Omron CX-Programmer project NewProject (CX-Programmer 9.61)

# PLC NewPLC1: CS1H-H CPU64
I/O table (CPU CS1H-CPU64H, CS1W-SCB21-V1): rack 0 slot 3 CS1W-AD081-V1; rack 0 slot 4 CS1W-CT041; rack 0 slot 5 CS1W-CT041; rack 0 slot 6 CS1W-DRM21-V1; rack 0 slot 8 CS1W-CLK21-V1; rack 0 slot 9 CS1W-ETN21(ETN21Mode); rack 1 slot 2 CS1W-MC221(-V1)

## Global symbols (name address type ; comment)
ALL_OK W303.15 BOOL
0.02 BOOL  ; DATA CLEAR
0.04 BOOL  ; CLEAR OF NG WORKPIECE INSULATION TEST
0.05 BOOL  ; CLEAR OF NG WORKPIECE IMPULSE MEASURE
0.06 BOOL  ; CLEAR OF NG WORKPIECE SWING MEASURE
0.07 BOOL  ; CLEAR OF NG WORKPIECE BEARING INSERT
0.08 BOOL  ; CLEAR OF NG WORKPIECE RESISTANCE MEASURE
0.09 BOOL  ; CLEAR OF NG WORKPIECE LENGTH MEASURE
0.10 BOOL  ; CLEAR OF LANE 1 CONFIRMATION THE OPERATION
0.11 BOOL  ; CLEAR OF LANE 2 CONFIRMATION THE OPERATION
0.12 BOOL  ; CLEAR OF ID INVALIDITY OPERATION
1001.04 BOOL  ; AUTO RUNNING (MACHINE No.1)
1001.05 BOOL  ; FAULT STOP AUX (MACHINE No.1)
1001.06 BOOL  ; FAULT STOP (MACHINE No.1)
1002.06 BOOL  ; AUTO RUNNING (MACHINE No.2)
1002.07 BOOL  ; FAULT STOP AUX (MACHINE No.2)
1002.08 BOOL  ; FAULT STOP (MACHINE No.2)
1005.00 BOOL  ; AUTO RUNNING (MACHINE No.3)
1005.01 BOOL  ; FAULT STOP AUX (MACHINE No.3)
1005.02 BOOL  ; FAULT STOP (MACHINE No.3)
1011.00 BOOL  ; AUTO RUNNING (MACHINE No.4)
1011.01 BOOL  ; FAULT STOP AUX (MACHINE No.4)
1011.02 BOOL  ; FAULT STOP (MACHINE No.4)
1011.03 BOOL  ; AUTO RUNNING (MACHINE No.5)
1011.04 BOOL  ; FAULT STOP AUX (MACHINE No.5)
1011.05 BOOL  ; FAULT STOP (MACHINE No.5)
1011.06 BOOL  ; AUTO RUNNING (MACHINE No.6)
1011.07 BOOL  ; FAULT STOP AUX (MACHINE No.6)
1011.08 BOOL  ; FAULT STOP (MACHINE No.6)
1013.04 BOOL  ; AUTO RUNNING (MACHINE No.7)
1013.05 BOOL  ; FAULT STOP AUX (MACHINE No.7)
1013.06 BOOL  ; FAULT STOP (MACHINE No.7)
1015.06 BOOL  ; AUTO RUNNING (MACHINE No.8)
1015.07 BOOL  ; FAULT STOP AUX (MACHINE No.8)
1015.08 BOOL  ; FAULT STOP (MACHINE No.8)
1016.08 BOOL  ; AUTO RUNNING (MACHINE No.9)
1016.09 BOOL  ; FAULT STOP AUX (MACHINE No.9)
1016.10 BOOL  ; FAULT STOP (MACHINE No.9)
1018.00 BOOL  ; CONVEYOR ROTATE FROM FORMER PROCESS
1019.06 BOOL  ; AUTO RUNNING (MACHINE No.10)
1019.07 BOOL  ; FAULT STOP AUX (MACHINE No.10)
1019.08 BOOL  ; FAULT STOP (MACHINE No.10)
1019.11 BOOL  ; from ball caulking mc  PROCESS, UNLOADING ST WORKPIECE NORMAL-TORQUE
1019.12 BOOL  ; From Ball Caulking, UNLOADING ST WORKPIECE NORMAL-TORQUE
1020.01 BOOL  ; ROTATION REQUEST TO FORMER PROCESS
1020.02 BOOL  ; ALL MACHINES SAVING ENERGY OF FLURESCENT LIGHT
1021.00 BOOL  ; AUTO RUNNING (MACHINE No.11)
1021.01 BOOL  ; FAULT STOP AUX (MACHINE No.11)
1021.02 BOOL  ; FAULT STOP (MACHINE No.11)
1200.00 BOOL  ; OFF IN EMERGENCY STOP
1200.01 BOOL  ; OFF IN AUTO STOP
1200.02 BOOL  ; OFF IN CYCLE STOP
1200.03 BOOL  ; OFF IN FAULT STOP
1200.04 BOOL  ; OFF IN TEMPORARY STOP 1
1200.05 BOOL  ; OFF IN STOP WARNING
1200.06 BOOL  ; OFF IN TEMPORARY STOP 2
1200.07 BOOL  ; OFF IN ONLY ALARM
1200.08 BOOL  ; ALARM CALL
1200.09 BOOL  ; STOP WARNING CALL
1200.10 BOOL  ; FORMER/LATTER PROCESS CONDITION WAITING
1200.11 BOOL  ; ALARM ONLY
1200.12 BOOL  ; BUZZER ON 1
1200.13 BOOL  ; ALARM RESET 1
1200.14 BOOL  ; BUZZER ON 2
1200.15 BOOL  ; ALARM RESET 2
1201.00 BOOL  ; UNUSUAL FAULT WITH LAST SCAN
1201.01 BOOL  ; WITH FAULT
1201.02 BOOL  ; ALL CH ENQUIRY COMPLETION
1201.03 BOOL  ; WITH FAULT IN 150CH
1201.04 BOOL  ; WITH FAULT IN 151CH
1201.05 BOOL  ; WITH FAULT IN 152CH
1201.06 BOOL  ; WITH FAULT IN 153CH
1201.07 BOOL  ; WITH FAULT IN 154CH
1201.08 BOOL  ; WITH FAULT IN 155CH
1201.09 BOOL  ; WITH FAULT IN 156CH
1201.10 BOOL  ; WITH FAULT IN 157CH
1201.11 BOOL  ; WITH FAULT IN 158CH
1201.12 BOOL  ; WITH FAULT IN 159CH
1201.13 BOOL  ; ENQUIRY IN PROGRESS WITH FAULT IN CH
1201.14 BOOL  ; WITH FAULT AUXILIARY
1201.15 BOOL  ; FAULT INDICATION CIRCUIT EFFECTIVE
1202.00 BOOL  ; CH EACH FAULT BIT 1
1202.01 BOOL  ; CH EACH FAULT BIT 2
1202.02 BOOL  ; CH EACH FAULT BIT 4
1202.03 BOOL  ; CH EACH FAULT BIT 8
1203.00 BOOL  ; FAULT ENQUIRY IN PROGRESS BIT 00
1203.01 BOOL  ; FAULT ENQUIRY IN PROGRESS BIT 01
1203.02 BOOL  ; FAULT ENQUIRY IN PROGRESS BIT 02
1203.03 BOOL  ; FAULT ENQUIRY IN PROGRESS BIT 03
1203.04 BOOL  ; FAULT ENQUIRY IN PROGRESS BIT 04
1203.05 BOOL  ; FAULT ENQUIRY IN PROGRESS BIT 05
1203.06 BOOL  ; FAULT ENQUIRY IN PROGRESS BIT 06
1203.07 BOOL  ; FAULT ENQUIRY IN PROGRESS BIT 07
1203.08 BOOL  ; FAULT ENQUIRY IN PROGRESS BIT 08
1203.09 BOOL  ; FAULT ENQUIRY IN PROGRESS BIT 09
1203.10 BOOL  ; FAULT ENQUIRY IN PROGRESS BIT 10
1203.11 BOOL  ; FAULT ENQUIRY IN PROGRESS BIT 11
1203.12 BOOL  ; FAULT ENQUIRY IN PROGRESS BIT 12
1203.13 BOOL  ; FAULT ENQUIRY IN PROGRESS BIT 13
1203.14 BOOL  ; FAULT ENQUIRY IN PROGRESS BIT 14
1203.15 BOOL  ; FAULT ENQUIRY IN PROGRESS BIT 15
1204.00 BOOL  ; ENQUIRY IN PROGRESS CH CODE 1
1204.01 BOOL  ; ENQUIRY IN PROGRESS CH CODE 2
1204.02 BOOL  ; ENQUIRY IN PROGRESS CH CODE 4
1204.03 BOOL  ; ENQUIRY IN PROGRESS CH CODE 8
1205.00 BOOL  ; SEARCHING IN FIRST HALF 10CH
1205.01 BOOL  ; SEARCHING IN SECOND HALF 10CH
1205.03 BOOL  ; WITH FAULT IN 160CH
1205.04 BOOL  ; WITH FAULT IN 161CH
1205.05 BOOL  ; WITH FAULT IN 162CH
1205.06 BOOL  ; WITH FAULT IN 163CH
1205.07 BOOL  ; WITH FAULT IN 164CH
1205.08 BOOL  ; WITH FAULT IN 165CH
1205.09 BOOL  ; WITH FAULT IN 166CH
1205.10 BOOL  ; WITH FAULT IN 167CH
1205.11 BOOL  ; WITH FAULT IN 168CH
1205.12 BOOL  ; WITH FAULT IN 169CH
1206.00 BOOL  ; ENQUIRY IN PROGRESS CH CODE 1
1206.01 BOOL  ; ENQUIRY IN PROGRESS CH CODE 2
1206.02 BOOL  ; ENQUIRY IN PROGRESS CH CODE 4
1206.03 BOOL  ; ENQUIRY IN PROGRESS CH CODE 8
1207.00 BOOL  ; FAULT RESET AUXILIARY
1207.01 BOOL  ; FAULT RESET START UP
1207.02 BOOL  ; START UP AUXILIARY
1207.03 BOOL  ; FAULT INDICATION REDUCTION
1208.00 BOOL  ; INDIVIDUAL SELECTION MEMORY
1208.01 BOOL  ; INDIVIDUAL SELECTION MEMORY RELEASE
1208.02 BOOL  ; INDIVIDUAL OPERATION EFFECTIVE AUXILIARY
1208.03 BOOL  ; INDIVIDUAL OPERATION CIRCUIT EFFECTIVE
1208.04 BOOL  ; OPERATION MODE CHANGE PULSE
1208.15 BOOL  ; MASTER ON PULSE
1211.00 BOOL  ; 01ST ALRAM SALL ARIA NO FAULT
1211.01 BOOL  ; 02ST ALRAM SALL ARIA NO FAULT
1211.02 BOOL  ; 03ST ALRAM SALL ARIA NO FAULT
1211.03 BOOL  ; 04ST ALRAM SALL ARIA NO FAULT
1211.04 BOOL  ; 05ST ALRAM SALL ARIA NO FAULT
1211.05 BOOL  ; 06ST ALRAM SALL ARIA NO FAULT
1211.06 BOOL  ; 07ST ALRAM SALL ARIA NO FAULT
1211.07 BOOL  ; 08ST ALRAM SALL ARIA NO FAULT
1211.08 BOOL  ; 09ST ALRAM SALL ARIA NO FAULT
1211.09 BOOL  ; 10ST ALRAM SALL ARIA NO FAULT
1211.10 BOOL  ; 11ST ALRAM SALL ARIA NO FAULT
1211.11 BOOL  ; 12ST ALRAM SALL ARIA NO FAULT
1211.12 BOOL  ; 13ST ALRAM SALL ARIA NO FAULT
1211.13 BOOL  ; 14ST ALRAM SALL ARIA NO FAULT
1211.14 BOOL  ; 15ST ALRAM SALL ARIA NO FAULT
1211.15 BOOL  ; 16ST ALRAM SALL ARIA NO FAULT
1212.00 BOOL  ; 01ST WARNING CALL ARIA NO FAULT
1212.01 BOOL  ; 02ST WARNING CALL ARIA NO FAULT
1212.02 BOOL  ; 03ST WARNING CALL ARIA NO FAULT
1212.03 BOOL  ; 04ST WARNING CALL ARIA NO FAULT
1212.04 BOOL  ; 05ST WARNING CALL ARIA NO FAULT
1212.05 BOOL  ; 06ST WARNING CALL ARIA NO FAULT
1212.06 BOOL  ; 07ST WARNING CALL ARIA NO FAULT
1212.07 BOOL  ; 08ST WARNING CALL ARIA NO FAULT
1212.08 BOOL  ; 09ST WARNING CALL ARIA NO FAULT
1212.09 BOOL  ; 10ST WARNING CALL ARIA NO FAULT
1212.10 BOOL  ; 11ST WARNING CALL ARIA NO FAULT
1212.11 BOOL  ; 12ST WARNING CALL ARIA NO FAULT
1212.12 BOOL  ; 13ST WARNING CALL ARIA NO FAULT
1212.13 BOOL  ; 14ST WARNING CALL ARIA NO FAULT
1212.14 BOOL  ; 15ST WARNING CALL ARIA NO FAULT
1212.15 BOOL  ; 16ST WARNING CALL ARIA NO FAULT
1213.00 BOOL  ; 17ST ALRAM SALL ARIA NO FAULT
1213.01 BOOL  ; 18ST ALRAM SALL ARIA NO FAULT
1213.02 BOOL  ; 19ST ALRAM SALL ARIA NO FAULT
1213.03 BOOL  ; 20ST ALRAM SALL ARIA NO FAULT
1214.00 BOOL  ; 17ST WARNING CALL ARIA NO FAULT
1214.01 BOOL  ; 18ST WARNING CALL ARIA NO FAULT
1214.02 BOOL  ; 19ST WARNING CALL ARIA NO FAULT
1214.03 BOOL  ; 20ST WARNING CALL ARIA NO FAULT
1222.01 BOOL  ; SEQUENCER NORMAL(CS1)
1230.00 BOOL  ; CONVEYOR ON
1235.00 BOOL  ; BEARING SUPPLY ROBOT MOTION PERMIT
1235.01 BOOL  ; BEARING HANGER UPWARD
1235.02 BOOL  ; BEARING SUPPLY ROBOT PROGRAM START
1235.03 BOOL  ; BEARING SUPPLY ROBOT FIXID POSITION RETURN
1235.05 BOOL  ; BEARING SUPPLY ROBOT FIXID POSITION RETURN
1235.06 BOOL  ; BEARING SUPPLY ROBOT TAKING-OUT POSITION START
1235.07 BOOL  ; BEARING TAKE OUT
1235.08 BOOL  ; BEARING SUPPLY ROBOT TAKING-OUT POSITION
1236 CHANNEL  ; BEARING SUPPLY ROBOT OUTPUT
1236.15 BOOL  ; BEARING SUPPLY ROBOT FIXID POSITION
1311.00 BOOL  ; UNLOADING ROBOT GOOD PRODUCT
1350.03 BOOL  ; MASTER SWITCH ON TRIGGER
1350.04 BOOL  ; MASTER SWITCH OFF TRIGGER
1350.11 BOOL  ; X AXIS SETTING SCREEN
1351.08 BOOL  ; FLASH MEMORY PRESERVATION TIMING
1352.00 BOOL  ; FORWARDING PERMISSION
1352.01 BOOL  ; MEMORY DRIVING END
1400.09 BOOL  ; MEMORY WITH SET VALUE CHANGE
1400.10 BOOL  ; WORKPIECE NUMBER CHANGE CHECK
1400.11 BOOL  ; WORKPIECE NUMBER SET UP PB ON
1400.12 BOOL  ; SETTING WORKPIECE NUMBER CHANGE PULSE
1400.13 BOOL  ; SETTING WORKPIECE NUMBER CHANGE
1400.14 BOOL  ; WORKPIECE NUMBER REGISTRATION SCREEN
1400.15 BOOL  ; WORKPIECE NUMBER REGISTRATION SCREEN PULSE
1401.08 BOOL  ; UNDER WORKPIECE NUMBER 1 DISPLAY
1401.09 BOOL  ; UNDER 1 OR LESS WORKPIECE NUMBER DISPLAY
1401.10 BOOL  ; UNDER WORKPIECE NUMBER 9 DISPLAY
1401.11 BOOL  ; UNDER 9 OR MORE WORKPIECE NUMBER DISPLAY
1402.00 BOOL  ; One set display (thickness of core)
1402.01 BOOL  ; One or less is displayed (thickness of core)
1402.02 BOOL  ; Two set display (thickness of core)
1402.03 BOOL  ; Two or less is displayed (thickness of core)
1402.04 BOOL  ; One set display (coil end)
1402.05 BOOL  ; One or less is displayed (coil end)
1402.06 BOOL  ; Two set display (coil end)
1402.07 BOOL  ; Two or less is displayed (coil end)
1402.08 BOOL  ; One set display (bearing insert)
1402.09 BOOL  ; One or less is displayed (bearing insert)
1402.10 BOOL  ; Two set display (bearing insert)
1402.11 BOOL  ; Two or less is displayed (bearing insert)
1403.03 BOOL  ; WITH SET VALUE CHANGE 1
1403.04 BOOL  ; WITH SET VALUE CHANGE 2
1404.01 BOOL  ; Can one product number flow
1404.02 BOOL  ; Can two product number flow
1404.03 BOOL  ; Can three product number flow
1404.04 BOOL  ; Can four product number flow
1404.05 BOOL  ; Can five product number flow
1404.06 BOOL  ; Can six product number flow
1404.07 BOOL  ; Can seven product number flow
1404.08 BOOL  ; Can eight product number flow
1404.09 BOOL  ; Can nine product number flow
1535.00 BOOL  ; The unit is abnormal
1535.06 BOOL  ; Node address repetition
1537.00 BOOL  ; Collation is abnormal
1537.01 BOOL  ; The composition is abnormal
1537.02 BOOL  ; Remote I/O communication abnormality
1537.04 BOOL  ; The scanning list data is illegal
1537.05 BOOL  ; Master function I/O refreshing is abnormal
2000.09 BOOL  ; WITHSTAND VOLTAGE TESTER INTERLOCK
2000.12 BOOL  ; SIGNAL TOWER RED
2000.13 BOOL  ; SIGNAL TOWER YELLOW
2000.14 BOOL  ; SIGNAL TOWER GREEN
2000.15 BOOL  ; ALARM
2001.00 BOOL  ; LOADING CONVEYOR PALLET SHIFT FORWARD
2001.01 BOOL  ; LOADING CONVEYOR PALLET SHIFT BACKWARD
2001.02 BOOL  ; LOADING CONVEYOR PALLET DISCHARGE FORWARD
2001.03 BOOL  ; LOADING CONVEYOR PALLET DISCHARGE BACKWARD
2001.04 BOOL  ; LOADER FORWARD
2001.05 BOOL  ; LOADER BACKWARD
2001.06 BOOL  ; LOADER DOWNWARD
2001.07 BOOL  ; LOADER UPWARD
2001.08 BOOL  ; TURN LOADER CHUCK TURN
2001.09 BOOL  ; TURN LOADER RECHUCK TURN
2001.10 BOOL  ; LOADER CHUCK CLAMP
2001.11 BOOL  ; LOADER CHUCK UNCLAMP
2001.12 BOOL  ; WORKPIECE PUSHER FORWARD
2001.14 BOOL  ; POSITIONING ARROW FORWARD
2002.00 BOOL  ; CONTACT PROBE IN RESISTANCE FORWARD
2002.01 BOOL  ; CONTACT PROBE IN RESISTANCE BACKWARD
2002.02 BOOL  ; CONTACT PROBE IN INPULSE FORWARD
2002.04 BOOL  ; WORKPIECE CLAMP DOWNWARD
2002.05 BOOL  ; WORKPIECE CLAMP UPWARD
2002.06 BOOL  ; TRANSFER CARRIER LIFT UPWARD
2002.07 BOOL  ; TRANSFER CARRIER LIFT DOWNWARD
2002.08 BOOL  ; SUB TRANSFER CARRIER LIFT UPWARD
2002.09 BOOL  ; SUB TRANSFER CARRIER LIFT DOWNWARD
2002.10 BOOL  ; TRANSFER CARRIER FORWARD
2002.11 BOOL  ; TRANSFER CARRIER BACKWARD
2002.12 BOOL  ; LENGTH MEASUREMENT FORWARD
2002.13 BOOL  ; LENGTH MEASUREMENT BACKWARD
2002.14 BOOL  ; Work Clamp DownWard
2002.15 BOOL  ; Work Clamp UpWard
2003.00 BOOL  ; BEARING INSERT (HIGH SPEED) FORWARD
2003.01 BOOL  ; BEARING INSERT (HIGH SPEED) BACKWARD
2003.02 BOOL  ; BEARING INSERT (HIGH PRESSURE) ON
2003.03 BOOL  ; BEARING INSERT (HIGH PRESSURE) OFF
2003.04 BOOL  ; BEARING SHUTTER DOWNWARD
2003.05 BOOL  ; BEARING SHUTTER UPWARD
2003.06 BOOL  ; BEARING GUIDE FORWARD
2003.07 BOOL  ; BEARING GUIDE BACKWARD
2003.08 BOOL  ; BEARING ESCAPE FORWARD
2003.09 BOOL  ; BEARING ESCAPE BACKWARD
2003.10 BOOL  ; BEARING TRANSFER UPWARD
2003.11 BOOL  ; BEARING TRANSFER DOWNWARD
2003.12 BOOL  ; BEARING PUSHER BACKWARD
2003.13 BOOL  ; BEARING PUSHER FORWARD
2003.14 BOOL  ; Work Clamp DownWard
2003.15 BOOL  ; Work Clamp UpWard
2004.00 BOOL  ; BEARING TRANSFER CARRIER FORWARD
2004.01 BOOL  ; BEARING TRANSFER CARRIER BACKWARD
2004.02 BOOL  ; BEARING HANGER FORWARD
2004.03 BOOL  ; BEARING HANGER BACKWARD
2004.04 BOOL  ; BEARING HANGER DOWNWARD
2004.05 BOOL  ; BEARING HANGER UPWARD
2004.06 BOOL  ; UNLOADING ROBOT CHUCK CLAMP
2004.07 BOOL  ; UNLOADING ROBOT CHUCK UNCLAMP
2004.08 BOOL  ; BEARING TRAY ESCAPE FORWARD
2004.09 BOOL  ; BEARING TRAY ESCAPE BACKWARD
2004.10 BOOL  ; BEARING TRAY STOPPER BACKWARD
2004.11 BOOL  ; BEARING TRAY STOPPER FORWARD
2004.12 BOOL  ; BEARING TRAY HOME POSITIONING FORWARD
2004.13 BOOL  ; BEARING TRAY HOME POSITIONING BACKWARD
2004.14 BOOL  ; BEARING TRAY EXCHANGE DOWNWARD
2004.15 BOOL  ; BEARING TRAY EXCHANGE UPWARD
2005.00 BOOL  ; TO RESISTANCE MEASUREMENT_BCD LOWER BYTE OUTPUT
2005.07 BOOL  ; COUNTER
2008.09 BOOL  ; DEFECT DISCHARGING CONVEYOR ON
2008.10 BOOL  ; INVERTER GOOD
2009.00 BOOL  ; LOADING CONVEYOR PALLET SHIFT FORWARD END
2009.01 BOOL  ; LOADING CONVEYOR PALLET SHIFT BACKWARD END
2009.02 BOOL  ; LOADING CONVEYOR PALLET DISCHARGE FORWARD END
2009.03 BOOL  ; LOADING CONVEYOR PALLET DISCHARGE FORWARD END
2009.04 BOOL  ; PALLET ON LOADING CONVEYOR
2009.05 BOOL  ; WORKPIECE ON LOADING CONVEYOR
2010.00 BOOL  ; LOADER FORWARD END
2010.01 BOOL  ; LOADER BACKWARD END
2010.02 BOOL  ; LOADER DOWNWARD END
2010.03 BOOL  ; LOADER UPWARD END
2010.04 BOOL  ; TURN LOADER CHUCK TURN END
2010.05 BOOL  ; TURN LOADER CHUCK RETURN END
2010.07 BOOL  ; LOADER CHUCK UNCLAMP END
2010.08 BOOL  ; PX_ LOADER DOWNWARD END
2010.12 BOOL  ; Contact Probe Lower Resistance Forward
2010.13 BOOL  ; Contact Probe Lower Resistance BackWard
2010.14 BOOL  ; Contact Probe Upper Resistance Forward
2010.15 BOOL  ; Contact Probe Upper Resistance Backward
2011.00 BOOL  ; TRANSFER CARRIER FORWARD END
2011.01 BOOL  ; TRANSFER CARRIER BACKWARD END
2011.02 BOOL  ; TRANSFER CARRIER LIFT UPWARD END
2011.03 BOOL  ; TRANSFER CARRIER LIFT DOWNWARD END
2011.04 BOOL  ; SUB TRANSFER CARRIER LIFT UPWARD END
2011.05 BOOL  ; SUB TRANSFER CARRIER LIFT DOWNWARD END
2011.06 BOOL  ; WORKPIECE PUSHER FORWARD END
2011.07 BOOL  ; WORKPIECE PUSHER BACKWARD END
2011.08 BOOL  ; THICKNESS OF CORE S
2011.09 BOOL  ; THICKNESS OF CORE L
2011.12 BOOL  ; Upper impulse probe forward end
2011.13 BOOL  ; Upper impulse probe receding end
2011.14 BOOL  ; Lower Impulse Probe FWD
2011.15 BOOL  ; Lower impulse probe receding end
2012.00 BOOL  ; POSITIONING ARROW FORWARD END
2012.02 BOOL  ; WORKPIECE CLAMP IN RESISTANCE DOWNWARD END
2012.03 BOOL  ; WORKPIECE CLAMP IN RESISTANCE UPWARD END
2012.04 BOOL  ; WORKPIECE CLAMP IN INPULSE DOWNWARD END
2012.05 BOOL  ; WORKPIECE CLAMP IN INPULSE UPWARD END
2012.06 BOOL  ; CONTACT PROBE IN RESISTANCE FORWARD END
2012.08 BOOL  ; CONTACT PROBE IN INPULSE FORWARD END
2012.10 BOOL  ; CONFIRM POSITIONING
2012.11 BOOL  ; COIL END S
2012.12 BOOL  ; COIL END L
2013.00 BOOL  ; BEARING INSERT (HIGH SPEED) FORWARD END
2013.01 BOOL  ; BEARING INSERT (HIGH SPEED) BACKWARD END
2013.02 BOOL  ; BEARING INSERT (HIGH PRESSURE) ON
2013.04 BOOL  ; BEARING SHUTTER DOWNWARD END
2013.05 BOOL  ; BEARING SHUTTER UPWARD END
2013.06 BOOL  ; BEARING GUIDE FORWARD END
2013.07 BOOL  ; BEARING GUIDE BACKWARD END
2013.08 BOOL  ; BEARING ESCAPE FORWARD END
2013.09 BOOL  ; BEARING ESCAPE BACKWARD END
2013.10 BOOL  ; BEARING TRANSFER UPWARD END
2013.11 BOOL  ; BEARING TRANSFER DOWNWARD END
2013.12 BOOL  ; BEARING PUSHER BACKWARD END
2013.13 BOOL  ; BEARING PUSHER FORWARD END
2013.14 BOOL  ; Bearing press-fit work holding down end
2013.15 BOOL  ; Bearing press-fit work presser rising end
2014.00 BOOL  ; BEARING TRANSFER CARRIER FORWARD END
2014.01 BOOL  ; BEARING TRANSFER CARRIER BACKWARD END
2014.02 BOOL  ; BEARING HANGER FORWARD END
2014.03 BOOL  ; BEARING HANGER BACKWARD END
2014.04 BOOL  ; BEARING HANGER DOWNWARD END
2014.05 BOOL  ; BEARING HANGER UPWARD END
2014.06 BOOL  ; BEARING CHECK (INSIDE AND OUTSIDE)
2014.07 BOOL  ; BEARING CONFIRM
2014.08 BOOL  ; BEARING (BEFOR INSERT)
2014.09 BOOL  ; FULL BEARING
2014.14 BOOL  ; Work Clamp Downword
2014.15 BOOL  ; Work Clamp Upword
2015.00 BOOL  ; LENGTH MEASUREMENT FORWARD END
2015.01 BOOL  ; LENGTH MEASUREMENT BACKWARD END
2015.03 BOOL  ; UNLOADING ROBOT CHUCK UNCLAMP END
2015.04 BOOL  ; WORKPIECE ON DEFECT DISCHARGING CONVEYOR
2015.05 BOOL  ; FULL WORKPIECES ON DEFECT DISCHARGING CONVEYOR
2015.06 BOOL  ; DEFECT DISCHARGING CONVEYOR PAEKING POSITION
2015.07 BOOL  ; CONTAINER
2016.08 BOOL  ; OUT SLAVE 0 FAULT IN COMMUNICATION
2016.09 BOOL  ; OUT SLAVE 1 FAULT IN COMMUNICATION
2016.10 BOOL  ; OUT SLAVE 2 FAULT IN COMMUNICATION
2016.11 BOOL  ; OUT SLAVE 3 FAULT IN COMMUNICATION
2016.12 BOOL  ; OUT SLAVE 4 FAULT IN COMMUNICATION
2016.13 BOOL  ; OUT SLAVE 5 FAULT IN COMMUNICATION
2016.14 BOOL  ; OUT SLAVE 6 FAULT IN COMMUNICATION
2016.15 BOOL  ; OUT SLAVE 7 FAULT IN COMMUNICATION
2017.08 BOOL  ; IN SLAVE 0 FAULT IN COMMUNICATION
2017.09 BOOL  ; IN SLAVE 1 FAULT IN COMMUNICATION
2017.10 BOOL  ; IN SLAVE 2 FAULT IN COMMUNICATION
2017.11 BOOL  ; IN SLAVE 3 FAULT IN COMMUNICATION
2017.12 BOOL  ; IN SLAVE 4 FAULT IN COMMUNICATION
2017.13 BOOL  ; IN SLAVE 5 FAULT IN COMMUNICATION
2017.14 BOOL  ; IN SLAVE 6 FAULT IN COMMUNICATION
2017.15 BOOL  ; IN SLAVE 7 FAULT IN COMMUNICATION
2018.08 BOOL  ; OUT SLAVE 8 FAULT IN COMMUNICATION
2018.09 BOOL  ; OUT SLAVE 9 FAULT IN COMMUNICATION
2018.10 BOOL  ; OUT SLAVE 10 FAULT IN COMMUNICATION
2018.11 BOOL  ; OUT SLAVE 11 FAULT IN COMMUNICATION
2018.12 BOOL  ; OUT SLAVE 12 FAULT IN COMMUNICATION
2018.13 BOOL  ; OUT SLAVE 13 FAULT IN COMMUNICATION
2018.14 BOOL  ; OUT SLAVE 14 FAULT IN COMMUNICATION
2018.15 BOOL  ; OUT SLAVE 15 FAULT IN COMMUNICATION
2019.08 BOOL  ; IN SLAVE 8 FAULT IN COMMUNICATION
2019.09 BOOL  ; IN SLAVE 9 FAULT IN COMMUNICATION
2019.10 BOOL  ; IN SLAVE 10 FAULT IN COMMUNICATION
2019.11 BOOL  ; IN SLAVE 11 FAULT IN COMMUNICATION
2019.12 BOOL  ; IN SLAVE 12 FAULT IN COMMUNICATION
2019.13 BOOL  ; IN SLAVE 13 FAULT IN COMMUNICATION
2019.14 BOOL  ; IN SLAVE 14 FAULT IN COMMUNICATION
2019.15 BOOL  ; IN SLAVE 15 FAULT IN COMMUNICATION
2020.00 BOOL  ; POSITIONING 1 BACKWARD
2020.01 BOOL  ; POSITIONING 1 FORWARD
2020.02 BOOL  ; POSITIONING 2 BACKWARD
2020.03 BOOL  ; POSITIONING 2 FORWARD
2020.04 BOOL  ; ESCAPE BEFOR PALLETIZING UPWARD
2020.05 BOOL  ; ESCAPE BEFOR PALLETIZING DOWNWARD
2020.06 BOOL  ; STOPPER BEFOR PALLETIZING UPWARD
2020.07 BOOL  ; STOPPER BEFOR PALLETIZING DOWNWARD
2020.08 BOOL  ; PALLETIZING STOPPER DOWNWARD
2020.09 BOOL  ; PALLETIZING STOPPER UPWARD
2020.10 BOOL  ; STACKING STOPPER DOWNWARD
2020.11 BOOL  ; STACKING STOPPER UPWARD
2020.12 BOOL  ; UNLOADING ESCAPE UPWARD
2020.13 BOOL  ; UNLOADING ESCAPE DOWNWARD
2020.14 BOOL  ; UNLOADING STOPPER DOWNWARD
2020.15 BOOL  ; UNLOADING STOPPER UPWARD
2021.00 BOOL  ; LIFTER DOWNWARD
2021.01 BOOL  ; LIFTER UPWARD
2021.02 BOOL  ; DROP GUARD BACKWARD
2021.03 BOOL  ; DROP GUARD FORWARD
2021.04 BOOL  ; PALLETIZING LIFTER DOWNWARD
2021.05 BOOL  ; PALLETIZING LIFTER UPWARD
2021.06 BOOL  ; PALLETIZING HOOK BACKWARD
2021.07 BOOL  ; PALLETIZING HOOK FORWARD
2021.08 BOOL  ; STACKING LIFTER DOWNWARD
2021.09 BOOL  ; STACKING LIFTER UPWARD
2021.10 BOOL  ; STACKING HOOK BACKWARD
2021.11 BOOL  ; STACKING HOOK FORWARD
2022.00 BOOL  ; LOADING CONVEYOR
2022.01 BOOL  ; PALLETIZING CONVEYOR
2022.02 BOOL  ; CONVEYOR AFTER PALLETIZING
2022.03 BOOL  ; EXCHANGE CONVEYOR CW
2022.04 BOOL  ; EXCHANGE CONVEYOR CCW
2022.05 BOOL  ; STACKING CONVEYOR
2022.06 BOOL  ; UNLOADING CONVEYOR 1
2022.07 BOOL  ; UNLOADING CONVEYOR 2
2023.00 BOOL  ; POSITIONING 1 BACKWARD
2023.01 BOOL  ; POSITIONING 1 FORWARD
2023.02 BOOL  ; POSITIONING 2 BACKWARD
2023.03 BOOL  ; POSITIONING 2 FORWARD
2023.04 BOOL  ; ESCAPE BEFOR PALLETIZING UPWARD
2023.05 BOOL  ; ESCAPE BEFOR PALLETIZING DOWNWARD
2023.06 BOOL  ; STOPPER BEFOR PALLETIZING UPWARD
2023.07 BOOL  ; STOPPER BEFOR PALLETIZING DOWNWARD
2023.08 BOOL  ; PALLETIZING STOPPER DOWNWARD
2023.09 BOOL  ; PALLETIZING STOPPER UPWARD
2023.10 BOOL  ; STACKING STOPPER DOWNWARD
2023.11 BOOL  ; STACKING STOPPER UPWARD
2023.12 BOOL  ; UNLOADING ESCAPE UPWARD
2023.13 BOOL  ; UNLOADING ESCAPE DOWNWARD
2023.14 BOOL  ; UNLOADING STOPPER DOWNWARD
2023.15 BOOL  ; UNLOADING STOPPER UPWARD
2024.00 BOOL  ; LIFTER DOWNWARD
2024.01 BOOL  ; LIFTER UPWARD
2024.02 BOOL  ; DROP GUARD BACKWARD
2024.03 BOOL  ; DROP GUARD FORWARD
2024.04 BOOL  ; PALLETIZING LIFTER DOWNWARD
2024.05 BOOL  ; PALLETIZING LIFTER UPWARD
2024.06 BOOL  ; PALLETIZING HOOK BACKWARD
2024.07 BOOL  ; PALLETIZING HOOK FORWARD
2024.08 BOOL  ; STACKING LIFTER DOWNWARD
2024.09 BOOL  ; STACKING LIFTER UPWARD
2024.10 BOOL  ; STACKING HOOK BACKWARD
2024.11 BOOL  ; STACKING HOOK FORWARD
2025.00 BOOL  ; LOADING CONVEYOR
2025.01 BOOL  ; PALLETIZING CONVEYOR
2025.02 BOOL  ; CONVEYOR AFTER PALLETIZING
2025.03 BOOL  ; EXCHANGE CONVEYOR CW
2025.04 BOOL  ; EXCHANGE CONVEYOR CCW
2025.05 BOOL  ; STACKING CONVEYOR
2025.06 BOOL  ; UNLOADING CONVEYOR 1
2025.07 BOOL  ; UNLOADING CONVEYOR 2
2028.00 BOOL  ; STOPPER BEFOR PALLETIZING UPWARD END
2028.01 BOOL  ; STOPPER BEFOR PALLETIZING DOWNWARD END
2028.02 BOOL  ; ESCAPE BEFOR PALLETIZING UPWARD END
2028.03 BOOL  ; ESCAPE BEFOR PALLETIZING DOWNWARD END
2028.04 BOOL  ; PALLETIZING STOPPER DOWNWARD END
2028.05 BOOL  ; PALLETIZING STOPPER UPWARD END
2028.06 BOOL  ; PALLETIZING LIFTER 1 DOWNWARD END
2028.07 BOOL  ; PALLETIZING LIFTER 1 INTERMEDIATE POSITION
2028.08 BOOL  ; PALLETIZING LIFTER 1 UPWARD END
2028.09 BOOL  ; PALLETIZING LIFTER 2 DOWNWARD END
2028.10 BOOL  ; PALLETIZING LIFTER 2 INTERMEDIATE POSITION
2028.11 BOOL  ; PALLETIZING LIFTER 2 UPWARD END
2028.12 BOOL  ; PALLETIZING HOOK 1 BACKWARD END
2028.13 BOOL  ; PALLETIZING HOOK 1 FORWARD END
2028.14 BOOL  ; PALLETIZING HOOK 2 BACKWARD END
2028.15 BOOL  ; PALLETIZING HOOK 2 FORWARD END
2029.00 BOOL  ; POSITIONING 2 BACKWARD END
2029.01 BOOL  ; POSITIONING 2 FORWARD END
2029.02 BOOL  ; POSITIONING 1 BACKWARD END
2029.03 BOOL  ; POSITIONING 1 FORWARD END
2029.04 BOOL  ; LOADING CONTAINER
2029.05 BOOL  ; CONTAINER BEFOR PALLETIZING
2029.06 BOOL  ; PALLETIZING CONTAINER
2029.07 BOOL  ; PALLETIZING CONTAINER UPPER SECTION
2029.08 BOOL  ; CONTAINER BEFOR EXCHANGE
2029.09 BOOL  ; EXCHANGE CONTAINER
2030.00 BOOL  ; LIFTER DOWNWARD END
2030.01 BOOL  ; LIFTER UPWARD END
2030.02 BOOL  ; DROP GUARD BACKWARD END
2030.03 BOOL  ; DROP GUARD FORWARD END
2030.04 BOOL  ; STACKING LIFTER 1 DOWNWARD END
2030.05 BOOL  ; STACKING LIFTER 1 INTERMEDIATE POSITION
2030.06 BOOL  ; STACKING LIFTER 1 UPWARD END
2030.07 BOOL  ; STACKING LIFTER 2 DOWNWARD END
2030.08 BOOL  ; STACKING LIFTER 2 INTERMEDIATE POSITION
2030.09 BOOL  ; STACKING LIFTER 2 UPWARD END
2030.10 BOOL  ; STACKING HOOK 1 BACKWARD END
2030.11 BOOL  ; STACKING HOOK 1 FORWARD END
2030.12 BOOL  ; STACKING HOOK 2 BACKWARD END
2030.13 BOOL  ; STACKING HOOK 2 FORWARD END
2030.14 BOOL  ; STACKING STOPPER DOWNWARD END
2030.15 BOOL  ; STACKING STOPPER UPWARD END
2031.00 BOOL  ; UNLOADING ESCAPE UPWARD END
2031.01 BOOL  ; UNLOADING ESCAPE DOWNWARD END
2031.02 BOOL  ; UNLOADING STOPPER DOWNWARD END
2031.03 BOOL  ; UNLOADING STOPPER UPWARD END
2031.04 BOOL  ; PASSING EXCHANGE CONTAINER
2031.05 BOOL  ; STACKING CONTAINER UPPER SECTION
2031.06 BOOL  ; STACKING CONTAINER
2031.07 BOOL  ; FULL CONTAINERS ON UNLOADING CONVEYOR
2031.08 BOOL  ; UNLOADING CONTAINERS
2032.00 BOOL  ; STOPPER BEFOR PALLETIZING UPWARD END
2032.01 BOOL  ; STOPPER BEFOR PALLETIZING DOWNWARD END
2032.02 BOOL  ; ESCAPE BEFOR PALLETIZING UPWARD END
2032.03 BOOL  ; ESCAPE BEFOR PALLETIZING DOWNWARD END
2032.04 BOOL  ; PALLETIZING STOPPER DOWNWARD END
2032.05 BOOL  ; PALLETIZING STOPPER UPWARD END
2032.06 BOOL  ; PALLETIZING LIFTER 1 DOWNWARD END
2032.07 BOOL  ; PALLETIZING LIFTER 1 INTERMEDIATE POSITION
2032.08 BOOL  ; PALLETIZING LIFTER 1 UPWARD END
2032.09 BOOL  ; PALLETIZING LIFTER 2 DOWNWARD END
2032.10 BOOL  ; PALLETIZING LIFTER 2 INTERMEDIATE POSITION
2032.11 BOOL  ; PALLETIZING LIFTER 2 UPWARD END
2032.12 BOOL  ; PALLETIZING HOOK 1 BACKWARD END
2032.13 BOOL  ; PALLETIZING HOOK 1 FORWARD END
2032.14 BOOL  ; PALLETIZING HOOK 2 BACKWARD END
2032.15 BOOL  ; PALLETIZING HOOK 2 FORWARD END
2033.00 BOOL  ; POSITIONING 2 BACKWARD END
2033.01 BOOL  ; POSITIONING 2 FORWARD END
2033.02 BOOL  ; POSITIONING 1 BACKWARD END
2033.03 BOOL  ; POSITIONING 1 FORWARD END
2033.04 BOOL  ; LOADING CONTAINER
2033.05 BOOL  ; CONTAINER BEFOR PALLETIZING
2033.06 BOOL  ; PALLETIZING CONTAINER
2033.07 BOOL  ; PALLETIZING CONTAINER UPPER SECTION
2033.08 BOOL  ; CONTAINER BEFOR EXCHANGE
2033.09 BOOL  ; EXCHANGE CONTAINER
2034.00 BOOL  ; LIFTER DOWNWARD END
2034.01 BOOL  ; LIFTER UPWARD END
2034.02 BOOL  ; DROP GUARD BACKWARD END
2034.03 BOOL  ; DROP GUARD FORWARD END
2034.04 BOOL  ; STACKING LIFTER 1 DOWNWARD END
2034.05 BOOL  ; STACKING LIFTER 1 INTERMEDIATE POSITION
2034.06 BOOL  ; STACKING LIFTER 1 UPWARD END
2034.07 BOOL  ; STACKING LIFTER 2 DOWNWARD END
2034.08 BOOL  ; STACKING LIFTER 2 INTERMEDIATE POSITION
2034.09 BOOL  ; STACKING LIFTER 2 UPWARD END
2034.10 BOOL  ; STACKING HOOK 1 BACKWARD END
2034.11 BOOL  ; STACKING HOOK 1 FORWARD END
2034.12 BOOL  ; STACKING HOOK 2 BACKWARD END
2034.13 BOOL  ; STACKING HOOK 2 FORWARD END
2034.14 BOOL  ; STACKING STOPPER DOWNWARD END
2034.15 BOOL  ; STACKING STOPPER UPWARD END
2035.00 BOOL  ; UNLOADING ESCAPE UPWARD END
2035.01 BOOL  ; UNLOADING ESCAPE DOWNWARD END
2035.02 BOOL  ; UNLOADING STOPPER DOWNWARD END
2035.03 BOOL  ; UNLOADING STOPPER UPWARD END
2035.04 BOOL  ; PASSING EXCHANGE CONTAINER
2035.05 BOOL  ; STACKING CONTAINER UPPER SECTION
2035.06 BOOL  ; STACKING CONTAINER
2035.07 BOOL  ; FULL CONTAINERS ON UNLOADING CONVEYOR
2035.08 BOOL  ; UNLOADING CONTAINERS
2036.08 BOOL  ; OUT SLAVE 0 FAULT IN COMMUNICATION
2036.09 BOOL  ; OUT SLAVE 1 FAULT IN COMMUNICATION
2036.10 BOOL  ; OUT SLAVE 2 FAULT IN COMMUNICATION
2036.11 BOOL  ; OUT SLAVE 3 FAULT IN COMMUNICATION
2036.12 BOOL  ; OUT SLAVE 4 FAULT IN COMMUNICATION
2036.13 BOOL  ; OUT SLAVE 5 FAULT IN COMMUNICATION
2036.14 BOOL  ; OUT SLAVE 6 FAULT IN COMMUNICATION
2036.15 BOOL  ; OUT SLAVE 7 FAULT IN COMMUNICATION
2037.08 BOOL  ; IN SLAVE 0 FAULT IN COMMUNICATION
2037.09 BOOL  ; IN SLAVE 1 FAULT IN COMMUNICATION
2037.10 BOOL  ; IN SLAVE 2 FAULT IN COMMUNICATION
2037.11 BOOL  ; IN SLAVE 3 FAULT IN COMMUNICATION
2037.12 BOOL  ; IN SLAVE 4 FAULT IN COMMUNICATION
2037.13 BOOL  ; IN SLAVE 5 FAULT IN COMMUNICATION
2037.14 BOOL  ; IN SLAVE 6 FAULT IN COMMUNICATION
2037.15 BOOL  ; IN SLAVE 7 FAULT IN COMMUNICATION
2038.08 BOOL  ; OUT SLAVE 8 FAULT IN COMMUNICATION
2038.09 BOOL  ; OUT SLAVE 9 FAULT IN COMMUNICATION
2038.10 BOOL  ; OUT SLAVE 10 FAULT IN COMMUNICATION
2038.11 BOOL  ; OUT SLAVE 11 FAULT IN COMMUNICATION
2038.12 BOOL  ; OUT SLAVE 12 FAULT IN COMMUNICATION
2038.13 BOOL  ; OUT SLAVE 13 FAULT IN COMMUNICATION
2038.14 BOOL  ; OUT SLAVE 14 FAULT IN COMMUNICATION
2038.15 BOOL  ; OUT SLAVE 15 FAULT IN COMMUNICATION
2039.08 BOOL  ; IN SLAVE 8 FAULT IN COMMUNICATION
2039.09 BOOL  ; IN SLAVE 9 FAULT IN COMMUNICATION
2039.10 BOOL  ; IN SLAVE 10 FAULT IN COMMUNICATION
2039.11 BOOL  ; IN SLAVE 11 FAULT IN COMMUNICATION
2039.12 BOOL  ; IN SLAVE 12 FAULT IN COMMUNICATION
2039.13 BOOL  ; IN SLAVE 13 FAULT IN COMMUNICATION
2039.14 BOOL  ; IN SLAVE 14 FAULT IN COMMUNICATION
2039.15 BOOL  ; IN SLAVE 15 FAULT IN COMMUNICATION
2040.00 BOOL  ; DEFECT DISCHARGING CONVEYOR START
2040.01 BOOL  ; DEFECT DISCHARGING CONVEYOR HIGH SPEED
2040.04 BOOL  ; DRIVE WORKPIECE
2040.05 BOOL  ; DRIVE WORKPIECE
2040.09 BOOL  ; FLURESCENT LIGHT OFF
2040.10 BOOL  ; DEFECT DISCHARGING CONVEYOR ON
2040.11 BOOL  ; LANE 1 UNLOADING
2040.12 BOOL  ; LANE 2 UNLOADING
2040.15 BOOL  ; Imagerogar 1
2041 CHANNEL  ; COMMAND POSITION
2041.00 BOOL  ; BEARING SUPPLY ROBOT HOLD
2041.01 BOOL  ; BEARING SUPPLY ROBOT SERVO ON
2041.02 BOOL  ; BEARING SUPPLY ROBOT RESET
2041.03 BOOL  ; BEARING SUPPLY ROBOT START
2042.00 BOOL  ; EXCHANGE CONVEYOR CW ROTATE
2042.01 BOOL  ; EXCHANGE CONVEYOR CCW ROTATE
2042.02 BOOL  ; LOADING CONVEYOR ON
2042.03 BOOL  ; UNLOADING CONVEYOR ON
2042.05 BOOL  ; Resistance Meas. Change Relay 6
2042.06 BOOL  ; Resistance Meas. Change Relay 12
2042.07 BOOL  ; Resistance Meas. Change Relay 13
2042.08 BOOL  ; Resistance Meas. Change Relay 13
2042.09 BOOL  ; Resistance Meas. Change Relay 14
2042.10 BOOL  ; Resistance Meas. Change Relay 15
2042.11 BOOL  ; Resistance Meas. Change Relay 16
2042.12 BOOL  ; Resistance Meas. Change Relay 16
2042.13 BOOL  ; Resistance Meas. Change Relay 17
2042.14 BOOL  ; Resistance Meas. Change Relay 15
2042.15 BOOL  ; Resistance Meas. Change Relay 2
2043.00 BOOL  ; WITH.VOL.MEAS. START
2043.01 BOOL  ; WITH.VOL.MEAS. STOP
2043.02 BOOL  ; RESISTANCE MEAS. TRIG
2043.09 BOOL  ; COUNTER
2043.10 BOOL  ; INPULSE DISPLAY OFF
2043.11 BOOL  ; INPULSE MEAS. START
2043.12 BOOL  ; INPULSE MEAS. RESET
2043.13 BOOL  ; INPULSE TRIG SIGNAL
2044 CHANNEL  ; IMPULSE TESTER
2044.09 BOOL  ; COUNTER
2045 CHANNEL  ; Impulse switching relay
2045.00 BOOL  ; WITHSTAND CIRCUIT CONNECTION
2045.01 BOOL  ; CONDUCTOT CHECK
2046 CHANNEL  ; IMPULSE RELAY
2047 CHANNEL  ; RESISTANCE MEASUREMENT CHANGE RELAY
2047.00 BOOL  ; Resistance Meas. Change Relay 1
2047.01 BOOL  ; Resistance Meas. Change Relay 2
2047.02 BOOL  ; Resistance Meas. Change Relay 3
2047.03 BOOL  ; Resistance Meas. Change Relay 4
2047.04 BOOL  ; Resistance Meas. Change Relay 5
2047.05 BOOL  ; Resistance Meas. Change Relay 6
2047.06 BOOL  ; Resistance Meas. Change Relay 7
2047.07 BOOL  ; Resistance Meas. Change Relay 8
2047.08 BOOL  ; Resistance Meas. Change Relay 9
2047.09 BOOL  ; Resistance Meas. Change Relay 10
2047.10 BOOL  ; Resistance Meas. Change Relay 11
2047.11 BOOL  ; Resistance Meas. Change Relay 12
2047.12 BOOL  ; Resistance Meas. Change Relay 13
2047.13 BOOL  ; Resistance Meas. Change Relay 14
2047.14 BOOL  ; Turn Number Description Switching Relay 1
2047.15 BOOL  ; Turn Number Description Switching Relay 1
2048.00 BOOL  ; INVERTER 2 GOOD
2048.02 BOOL  ; LANE 1 UNLOADING START
2048.03 BOOL  ; ﾚｰﾝ2排出部起動PB
2048.05 BOOL  ; ROBOT CPU GOOD
2048.06 BOOL  ; LANE 1 UNLOADING START
2048.07 BOOL  ; LANE 2 UNLOADING START
2048.08 BOOL  ; DEFECT DISCHARGING CONVEYOR START
2048.09 BOOL  ; ADD SENSOR CHECK BEARING
2049 CHANNEL  ; BEARING SUPPLY ROBOT OUTPUT
2049.00 BOOL  ; BEARING SUPPLY ROBOT MOTION
2049.02 BOOL  ; BEARING SUPPLY ROBOT ALARM
2049.04 BOOL  ; BEARING SUPPLY ROBOT HOMING COMPLETE
2049.05 BOOL  ; BEARING SUPPLY ROBOT POSITIONING COMPLETE
2049.06 BOOL  ; BEARING SUPPLY ROBOT SERVO ON
2051 CHANNEL  ; RESISTANCE MEASUREMENT DATA BCD
2051.00 BOOL  ; RESISTANCE MEASURED VALUE BCD4-0/RNG_OUT0
2051.01 BOOL  ; RESISTANCE MEASURED VALUE BCD4-1 /RNG_OUT1
2051.02 BOOL  ; RESISTANCE MEASURED VALUE BCD4-2 /RNG_OUT2
2051.03 BOOL  ; RESISTANCE MEASURED VALUE BCD4-3 /RNG_OUT3
2051.04 BOOL  ; RESISTANCE MEASURED VALUE BCD5/BCD1-0
2051.05 BOOL  ; RESISTANCE MEASURED VALUE BCD5/BCD1-1
2051.06 BOOL  ; RESISTANCE MEASURED VALUE BCD5/BCD1-2
2051.07 BOOL  ; RESISTANCE MEASURED VALUE BCD5/BCD1-3
2051.08 BOOL  ; RESISTANCE MEASURED VALUE BCD6/BCD2-0
2051.09 BOOL  ; RESISTANCE MEASURED VALUE BCD6/BCD2-1
2051.10 BOOL  ; RESISTANCE MEASURED VALUE BCD6/BCD2-2
2051.11 BOOL  ; RESISTANCE MEASURED VALUE BCD6/BCD2-3
2051.12 BOOL  ; RESISTANCE MEASURED VALUE BCD7/BCD3-0
2051.13 BOOL  ; RESISTANCE MEASURED VALUE BCD7/BCD3-1
2051.14 BOOL  ; RESISTANCE MEASURED VALUE BCD7/BCD3-2
2051.15 BOOL  ; RESISTANCE MEASURED VALUE BCD7/BCD3-3
2052 CHANNEL  ; RESISTANCE MEASUREMENT DATA BCD
2052.05 BOOL  ; RESISTANCE MEAS.1 ERR
2052.06 BOOL  ; RESISTANCE MEAS.1 INDEX
2052.07 BOOL  ; RESISTANCE MEAS.1 EOC
2052.08 BOOL  ; RESISTANCE MEAS.1 BCD 10^4X1
2052.09 BOOL  ; RESISTANCE MEAS.1 BCD 10^4X2
2052.10 BOOL  ; RESISTANCE MEAS.1 BCD 10^4X4
2052.13 BOOL  ; RESISTANCE MEAS.1 BCD 10^5X2
2052.14 BOOL  ; RESISTANCE MEAS.1 BCD 10^5X4
2052.15 BOOL  ; RESISTANCE MEAS.1 BCD 10^5X8
2053.00 BOOL  ; WITH.VOL.TEST
2053.01 BOOL  ; WITH.VOL.OK
2053.02 BOOL  ; WITH.VOL.HIGH-FAULT
2053.03 BOOL  ; WITH.VOL.LOW-FAULT
2053.04 BOOL  ; WITH.VOL.READY
2053.05 BOOL  ; WITH.VOL.PROTECTION
2053.06 BOOL  ; $?St$Bk?_#[5] / NUMBER OF TURNS "HI"$?St$Bk?_#[5]
2053.07 BOOL  ; $?St$Bk?_#[6] / NUMBER OF TURNS "IN"$?St$Bk?_#[6]
2053.08 BOOL  ; $?St$Bk?_#[7] / NUMBER OF TURNS "LO"$?St$Bk?_#[7]
2053.09 BOOL  ; EOM
2053.12 BOOL  ; INPULSE TESTER 1 BUSY
2053.13 BOOL  ; INPULSE TESTER 1 OK
2053.14 BOOL  ; INPULSE TESTER 1 NG
2053.15 BOOL  ; INPULSE TESTER 1 ERROR
2056.08 BOOL  ; OUT SLAVE 0 FAULT IN COMMUNICATION
2056.09 BOOL  ; OUT SLAVE 1 FAULT IN COMMUNICATION
2056.10 BOOL  ; OUT SLAVE 2 FAULT IN COMMUNICATION
2056.11 BOOL  ; OUT SLAVE 3 FAULT IN COMMUNICATION
2056.12 BOOL  ; OUT SLAVE 4 FAULT IN COMMUNICATION
2056.13 BOOL  ; OUT SLAVE 5 FAULT IN COMMUNICATION
2056.14 BOOL  ; OUT SLAVE 6 FAULT IN COMMUNICATION
2056.15 BOOL  ; OUT SLAVE 7 FAULT IN COMMUNICATION
2057.08 BOOL  ; IN SLAVE 0 FAULT IN COMMUNICATION
2057.09 BOOL  ; IN SLAVE 1 FAULT IN COMMUNICATION
2057.10 BOOL  ; IN SLAVE 2 FAULT IN COMMUNICATION
2057.11 BOOL  ; IN SLAVE 3 FAULT IN COMMUNICATION
2057.12 BOOL  ; IN SLAVE 4 FAULT IN COMMUNICATION
2057.13 BOOL  ; IN SLAVE 5 FAULT IN COMMUNICATION
2057.14 BOOL  ; IN SLAVE 6 FAULT IN COMMUNICATION
2057.15 BOOL  ; IN SLAVE 7 FAULT IN COMMUNICATION
2058.08 BOOL  ; OUT SLAVE 8 FAULT IN COMMUNICATION
2058.09 BOOL  ; OUT SLAVE 9 FAULT IN COMMUNICATION
2058.10 BOOL  ; OUT SLAVE 10 FAULT IN COMMUNICATION
2058.11 BOOL  ; OUT SLAVE 11 FAULT IN COMMUNICATION
2058.12 BOOL  ; OUT SLAVE 12 FAULT IN COMMUNICATION
2058.13 BOOL  ; OUT SLAVE 13 FAULT IN COMMUNICATION
2058.14 BOOL  ; OUT SLAVE 14 FAULT IN COMMUNICATION
2058.15 BOOL  ; OUT SLAVE 15 FAULT IN COMMUNICATION
2059.08 BOOL  ; IN SLAVE 8 FAULT IN COMMUNICATION
2059.09 BOOL  ; IN SLAVE 9 FAULT IN COMMUNICATION
2059.10 BOOL  ; IN SLAVE 10 FAULT IN COMMUNICATION
2059.11 BOOL  ; IN SLAVE 11 FAULT IN COMMUNICATION
2059.12 BOOL  ; IN SLAVE 12 FAULT IN COMMUNICATION
2059.13 BOOL  ; IN SLAVE 13 FAULT IN COMMUNICATION
2059.14 BOOL  ; IN SLAVE 14 FAULT IN COMMUNICATION
2059.15 BOOL  ; IN SLAVE 15 FAULT IN COMMUNICATION
2061 CHANNEL  ; INPUT 1 CONVERSION VALUE
2069.00 BOOL  ; INPUT 1 DISCONNECTION DETECTION
2080.00 BOOL  ; MASTER ON PERMISSION
2080.01 BOOL  ; SAFETY DOOR OPEN OK(FROM PLC)
2080.02 BOOL  ; CONVEYOR ON PERMISSION
2080.03 BOOL  ; CONVEYOR ECO RUNNING 1
2080.04 BOOL  ; MASTER SWITCH ON
2080.05 BOOL  ; CONVEYOR SWITCH ON
2080.06 BOOL  ; CONVEYOR ECO RUNNING 2
2080.07 BOOL  ; ROBOT STOP FROM PLC(AT OFF)
2088.00 BOOL  ; BEARING TRAY EXCHANGE DOWNWARD END
2088.01 BOOL  ; BEARING TRAY EXCHANGE UPWARD END
2088.02 BOOL  ; BEARING TRAY HOME POSITIONING BACKWARD END
2088.03 BOOL  ; BEARING TRAY HOME POSITIONING FORWARD END
2088.04 BOOL  ; BEARING TRAY STOPPER BACKWARD END
2088.05 BOOL  ; BEARING TRAY STOPPER FORWARD END
2088.06 BOOL  ; BEARING TRAY ESCAPE FORWARD END
2088.07 BOOL  ; BEARING TRAY ESCAPE BACKWARD END
2088.08 BOOL  ; LOADING BEARING TRAY
2088.09 BOOL  ; BEARING TRAY BEFOR EXCHANGE
2088.10 BOOL  ; EXCHANGE BEARING TRAY
2088.11 BOOL  ; PASSING BEARING TRAY
2088.12 BOOL  ; PASSING UNLOADING BEARING TRAY
2090.00 BOOL  ; FUSE GOOD
2090.01 BOOL  ; THERMAL RELAY GOOD
2090.02 BOOL  ; SAFETY CONFIRM 1-1(SAFETY DOOR SWITCH 1 CLOSE WHEN TEACHING ROBOT)
2090.03 BOOL  ; EX. HANDLE CONFIRMATION
2090.04 BOOL  ; SAFETY CONFIRM 2-1(SAFETY DOOR SWITCH 1 OPEN WHEN TEACHING ROBOT)
2090.05 BOOL  ; AIR CONFIRMATION
2090.06 BOOL  ; CONVEYOR THERMAL RELAY GOOD
2090.07 BOOL  ; MASTER ON CONFIRM
2090.08 BOOL  ; CONVEYOR ON CONFIRM
2090.09 BOOL  ; SAFETY CONFIRM 1-2(SAFETY DOOR SWITCH 2 CLOSE WHEN TEACHING ROBOT)
2090.10 BOOL  ; SAFETY CONFIRM 2-2(SAFETY DOOR SWITCH 2 OPEN WHEN TEACHING ROBOT)
2090.11 BOOL  ; SAFTY CONFIRM INVALID(KEY SWITCH TEACH ON)
2090.12 BOOL  ; EMERGENCY STOP PUSH BUTTON SWITCH OFF
2090.13 BOOL  ; SAFTY CONFIRM INVALID PL
2090.14 BOOL  ; MASTER ON COND.(EXT. A SAFEGUARD)
2090.15 BOOL  ; OPERATION PANEL SURE PUSH BUTTON SWITCH
2091.07 BOOL  ; MASTER ON CONFIRM MC-A
2091.15 BOOL  ; OPERATION PANEL SURE PUSH BUTTON SWITCH CR-A
2096.08 BOOL  ; OUT SLAVE 0 FAULT IN COMMUNICATION
2096.09 BOOL  ; OUT SLAVE 1 FAULT IN COMMUNICATION
2096.10 BOOL  ; OUT SLAVE 2 FAULT IN COMMUNICATION
2096.11 BOOL  ; OUT SLAVE 3 FAULT IN COMMUNICATION
2096.12 BOOL  ; OUT SLAVE 4 FAULT IN COMMUNICATION
2096.13 BOOL  ; OUT SLAVE 5 FAULT IN COMMUNICATION
2096.14 BOOL  ; OUT SLAVE 6 FAULT IN COMMUNICATION
2096.15 BOOL  ; OUT SLAVE 7 FAULT IN COMMUNICATION
2097.08 BOOL  ; IN SLAVE 0 FAULT IN COMMUNICATION
2097.09 BOOL  ; IN SLAVE 1 FAULT IN COMMUNICATION
2097.10 BOOL  ; IN SLAVE 2 FAULT IN COMMUNICATION
2097.11 BOOL  ; IN SLAVE 3 FAULT IN COMMUNICATION
2097.12 BOOL  ; IN SLAVE 4 FAULT IN COMMUNICATION
2097.13 BOOL  ; IN SLAVE 5 FAULT IN COMMUNICATION
2097.14 BOOL  ; IN SLAVE 6 FAULT IN COMMUNICATION
2097.15 BOOL  ; IN SLAVE 7 FAULT IN COMMUNICATION
2098.08 BOOL  ; OUT SLAVE 8 FAULT IN COMMUNICATION
2098.09 BOOL  ; OUT SLAVE 9 FAULT IN COMMUNICATION
2098.10 BOOL  ; OUT SLAVE 10 FAULT IN COMMUNICATION
2098.11 BOOL  ; OUT SLAVE 11 FAULT IN COMMUNICATION
2098.12 BOOL  ; OUT SLAVE 12 FAULT IN COMMUNICATION
2098.13 BOOL  ; OUT SLAVE 13 FAULT IN COMMUNICATION
2098.14 BOOL  ; OUT SLAVE 14 FAULT IN COMMUNICATION
2098.15 BOOL  ; OUT SLAVE 15 FAULT IN COMMUNICATION
2099.08 BOOL  ; IN SLAVE 8 FAULT IN COMMUNICATION
2099.09 BOOL  ; IN SLAVE 9 FAULT IN COMMUNICATION
2099.10 BOOL  ; IN SLAVE 10 FAULT IN COMMUNICATION
2099.11 BOOL  ; IN SLAVE 11 FAULT IN COMMUNICATION
2099.12 BOOL  ; IN SLAVE 12 FAULT IN COMMUNICATION
2099.13 BOOL  ; IN SLAVE 13 FAULT IN COMMUNICATION
2099.14 BOOL  ; IN SLAVE 14 FAULT IN COMMUNICATION
2099.15 BOOL  ; IN SLAVE 15 FAULT IN COMMUNICATION
2100.00 BOOL  ; $?St$Bk?_#[8] / Brake / Output $?St$Bk?_#[8]
2100.14 BOOL  ; Error Reset Bit
2101.01 BOOL  ; OPTIONAL INPUT # 1
2101.02 BOOL  ; OPTIONAL INPUT # 2
2102 CHANNEL  ; Task 1 program number
2103.01 BOOL  ; Automatic/Manual Mode ↑
2103.02 BOOL  ; Cycle Start Bit
2103.03 BOOL  ; Single Block
2103.04 BOOL  ; Forced Block End
2103.05 BOOL  ; Pause
2103.06 BOOL  ; M Code Reset Bit
2103.07 BOOL  ; $?St$Bk?_#[9] / Program Number Read / Bit$?St$Bk?_#[9]
2103.09 BOOL  ; Teaching Bit
2103.10 BOOL  ; Teaching Type Bit
2106 CHANNEL  ; X AXIS OVERRIDE
2107.00 BOOL  ; Deceleration Stop
2107.01 BOOL  ; Origin Search
2107.02 BOOL  ; Reference Origin Return
2107.03 BOOL  ; Jogging
2107.04 BOOL  ; Error Counter Reset
2107.05 BOOL  ; Forced Origin
2107.06 BOOL  ; Absolute Origin Set
2107.08 BOOL  ; $?St$Bk?_#[10] / Enable MPG/Sync / Encoder$?St$Bk?_#[10]
2107.09 BOOL  ; Servo-lock
2107.10 BOOL  ; Servo-unlock
2107.11 BOOL  ; Driver Alarm Reset
2107.12 BOOL  ; Override Setting
2107.13 BOOL  ; Jog direction
2107.14 BOOL  ; $?St$Bk?_#[11] / MPG/Sync Encoder Ratio / Specifier 1$?St$Bk?_#[11]
2107.15 BOOL  ; $?St$Bk?_#[12] / MPG/Sync Encoder Ratio / Specifier 2$?St$Bk?_#[12]
2110.11 BOOL  ; TEACHING EFFECTIVE MODE INSIDE
2110.12 BOOL  ; TEACHING OCCUPATION MODE INSIDE
2110.14 BOOL  ; THE ERROR IS OCCURRING
2115.00 BOOL  ; Task Error Flag
2115.02 BOOL  ; Automatic Mode Flag
2115.03 BOOL  ; Manual Mode Flag
2115.04 BOOL  ; Program Execution Flag
2115.05 BOOL  ; $?St$Bk?_#[13] / Program Execution / Completed Flag$?St$Bk?_#[13]
2115.06 BOOL  ; Optional Input Standby
2115.07 BOOL  ; M Code Reset Standby
2115.08 BOOL  ; M Strobe
2115.09 BOOL  ; Cycle Start Received
2115.13 BOOL  ; Teaching Completed
2115.14 BOOL  ; Teaching Error
2115.15 BOOL  ; Teaching Address Over
2120 CHANNEL  ; PRESENT VALUE
2122.00 BOOL  ; Reference Origin
2122.01 BOOL  ; Busy Flag
2122.02 BOOL  ; Servo-lock ON
2122.03 BOOL  ; No Origin Flag
2122.04 BOOL  ; Axis Operating
2122.05 BOOL  ; Positioning Completed
2122.06 BOOL  ; Error Counter Warning
2122.07 BOOL  ; Alarm Input
2122.08 BOOL  ; Transfer Carrier FWD
2122.09 BOOL  ; Transfer Carrier BWD
2125.02 BOOL  ; Y AXIS BUSY FLAG
2202.00 BOOL  ; One high-speed counter opening gate
2202.01 BOOL  ; One high-speed counter close gate
2202.03 BOOL  ; One high-speed counter reset
2208.00 BOOL  ; Three high-speed counter opening gate
2208.01 BOOL  ; Three high-speed counter close gate
2208.03 BOOL  ; Three high-speed counter resets
2222 CHANNEL  ; One high-speed counter count value
2224.02 BOOL  ; One driving of a high-speed counter
2224.05 BOOL  ; One high-speed counter reset flag
2232 CHANNEL  ; Three high-speed counter count value
2234.02 BOOL  ; Three driving of a high-speed counter
2234.05 BOOL  ; Three high-speed counter reset flag
2242.00 BOOL  ; High-speed counter 1 opening gate
2242.01 BOOL  ; High-speed counter 1 close gate
2242.02 BOOL  ; High-speed counter 1 preset
2243 CHANNEL  ; One high-speed counter Priset value
2248.00 BOOL  ; High-speed counter 3 opening gate
2248.01 BOOL  ; High-speed counter 3 close gate
2248.02 BOOL  ; High-speed counter 3 preset
2249 CHANNEL  ; Three high-speed counter Priset value
2262 CHANNEL  ; One high-speed counter count value
2264.02 BOOL  ; Flag when one high-speed counter driving
2264.04 BOOL  ; One high-speed counter Prisettofrag
2272 CHANNEL  ; Three high-speed counter count value
2274.02 BOOL  ; Flag when three high-speed counter driving
2274.04 BOOL  ; Three high-speed counter Prisettofrag
3200 CHANNEL  ; DATA AREA 1
3200.00 BOOL  ; STEP STOP(ALL TASKS)
3200.02 BOOL  ; INSTANT STOP(ALL TASKS)
3200.03 BOOL  ; STROBE SIGNAL
3200.07 BOOL  ; COMMAND DATA(ODD PARITY)
3201 CHANNEL  ; DATA AREA 2
3202 CHANNEL  ; COMMAND AREA
3202.08 BOOL  ; input 552_GRIPPER CLAMP CONFIRM
3202.09 BOOL  ; input 553_GRIPPER UNCLAMP CONFIRM
3202.10 BOOL  ; input 554_LOADING WORKPIECE
3202.11 BOOL  ; input 555_POSITION NUMBER READING START
3203 CHANNEL  ; Position number
3210 CHANNEL  ; 書込みﾃﾞｰﾀ
3211 CHANNEL  ; ID読出開始ｱﾄﾞﾚｽ転送
3211.14 BOOL  ; Ｒ／Ｗ
3211.15 BOOL  ; トリガ
3212 CHANNEL  ; Writing data
3213 CHANNEL  ; READING START ADDRESS
3213.14 BOOL  ; READ / WRITE
3213.15 BOOL  ; TRIGGER
3214 CHANNEL  ; Writing data
3215 CHANNEL  ; READING START ADDRESS
3215.14 BOOL  ; READ / WRITE
3215.15 BOOL  ; TRIGGER
3216 CHANNEL  ; Writing data
3217 CHANNEL  ; READING START ADDRESS
3217.14 BOOL  ; READ / WRITE
3217.15 BOOL  ; TRIGGER
3250 CHANNEL  ; DATA AREA 1
3251 CHANNEL  ; DATA AREA 2
3252 CHANNEL  ; COMMAND AREA
3253 CHANNEL  ; RB1_Position number
3300.01 BOOL  ; ROBOT RUNNING
3300.02 BOOL  ; ROBOT FAULT
3300.03 BOOL  ; SERVO ON
3300.04 BOOL  ; ROBOT READY
3300.05 BOOL  ; Automatic mode
3300.06 BOOL  ; External mode
3300.07 BOOL  ; The battery remainder amount warning
3300.08 BOOL  ; ROBOT ALARM
3300.14 BOOL  ; Command processing completion
3301 CHANNEL  ; Status area
3302.00 BOOL  ; output 800_FIXED POSITION/ HOME POSITION
3302.02 BOOL  ; output 802
3302.03 BOOL  ; output 803_WORKPIECE LOADING SIGNAL
3302.04 BOOL  ; output 804_CHUCK CLAMP OUTPUT ON
3302.05 BOOL  ; output 805_UNCHUCK CLAMP OUTPUT ON
3302.06 BOOL  ; output 806_READING COMPLETION OF POSITION NUMBER
3310 CHANNEL  ; ID読出ﾃﾞｰﾀ
3311.13 BOOL  ; NG
3311.14 BOOL  ; NORMAL
3311.15 BOOL  ; HS
3312 CHANNEL  ; Reeding data of ID
3313.13 BOOL  ; NG
3313.14 BOOL  ; NORMAL
3313.15 BOOL  ; HS
3314 CHANNEL  ; Reeding data of ID
3315.13 BOOL  ; NG
3315.14 BOOL  ; NORMAL
3315.15 BOOL  ; HS
3316 CHANNEL  ; Reeding data of ID
3317.13 BOOL  ; NG
3317.14 BOOL  ; NORMAL
3317.15 BOOL  ; HS
3800.00 BOOL  ; SURE PUSH BUTTON SWITCH ON
3800.01 BOOL  ; AUTO RUN CONDITION
3800.02 BOOL  ; NO CYCLE
3800.05 BOOL  ; AUTO RUNNING
3800.06 BOOL  ; AUTO START PULSE
3800.07 BOOL  ; AUTO STOP PULSE
3800.10 BOOL  ; WORKPIECE LOADING STOP
3800.11 BOOL  ; FINISHING OPERATION COMPLETION AND NO WORKPIECES
3800.12 BOOL  ; THERE IS NO WORK IN EQUIPMENT
3800.13 BOOL  ; Tray discharge Operation Running Complete
3800.14 BOOL  ; Trar Discharge Complete
3800.15 BOOL  ; Completion at in-flight all ST cycle
3801.00 BOOL  ; AUTO RUNNING(RESTART)
3801.10 BOOL  ; TEMPORARY STOP OPERATION EFFECTIVE
3801.12 BOOL  ; During master check
3801.13 BOOL  ; Masterwork in-flight capture completed
3803.10 BOOL  ; 前工程より作業終了ﾌﾗｸﾞ確認
3803.14 BOOL  ; Master check abnormality confirmation
3803.15 BOOL  ; Master check completed
3805.01 BOOL  ; Tip runout master check OK
3805.02 BOOL  ; Woom swing master check OK
3805.03 BOOL  ; Resistance 1 master check OK
3805.04 BOOL  ; Resistance 2 Master check OK
3805.05 BOOL  ; Resistance 3 Master Check OK
3805.06 BOOL  ; Resistance 4 Master Check OK
3805.07 BOOL  ; Impals 1 Master Check OK
3805.08 BOOL  ; Impals 2 Master Check OK
3805.09 BOOL  ; Impals 3 Master Check OK
3805.10 BOOL  ; 耐圧ﾏｽﾀｰﾁｪｯｸOK
3805.13 BOOL  ; Electric check master check completion memory
3805.14 BOOL  ; Abnormal stop before completion of electric check master check
3805.15 BOOL  ; Electric check master check completed
3806.00 BOOL  ; 寸法ﾏｽﾀ合わせﾓｰﾄﾞ(LM)完了
3806.01 BOOL  ; Dimension Master Check Mode (LM) Completed
3806.02 BOOL  ; Dimension master alignment mode (S) completed
3806.03 BOOL  ; Dimension master check mode (S) completed
3806.05 BOOL  ; Dimension master alignment mode (LM) completion memory
3806.06 BOOL  ; Dimension master alignment mode (S) completion memory
3806.10 BOOL  ; 自動切り1Scan遅れ
3806.12 BOOL  ; Forced descent operation ON during master check
3807.00 BOOL  ; Master Zero Complete
3807.01 BOOL  ; Dimension measurement + NG master check OK
3807.02 BOOL  ; Dimension measurement-NG master check OK
3807.05 BOOL  ; Maser Check Start
3807.13 BOOL  ; Dimension master check abnormality temporary memory
3807.14 BOOL  ; Master check abnormality (dimensions)
3807.15 BOOL  ; Master check completed (dimensions)
3808.12 BOOL  ; During master check (dimensions)
3808.13 BOOL  ; Dimension measurement master check completion memory
3808.14 BOOL  ; Dimension measurement Stop abnormality before completion of master check
3808.15 BOOL  ; Dimension measurement master check completed
3810 CHANNEL  ; Master check result flag
3810.01 BOOL  ; ROBOT START CONDITION
3810.02 BOOL  ; ROBOT PREPARATION START
3810.04 BOOL  ; I/O COMMAND CLEAR_1 SCAN TIMING
3810.05 BOOL  ; MODE CHANGE MOTOR ON->CAL->SP100->EXTERNAL MODE
3810.06 BOOL  ; COMPLETION OF ROBOT MODE CHANGE
3810.07 BOOL  ; FIXED POSITION RETURN PB ON
3810.09 BOOL  ; WITH FIXED POSITION RETURN OPERATION
3810.10 BOOL  ; FIXED POSITION RETURN NO OPERATION
3810.11 BOOL  ; FIXED POSITION RETURN OPERATION CONDITION
3810.12 BOOL  ; FIXED POSITION RETURN PROGRAM START
3810.13 BOOL  ; FIXED POSITION RETURN PROGRAM START RESET
3810.14 BOOL  ; INTERFERENCE
3810.15 BOOL  ; COMPLETION CLEAR PULSE ROBOT PREPARATION
3811.00 BOOL  ; COMPLETION AUXILIARY ROBOT PREPARATION
3811.01 BOOL  ; COMPLETION OF ROBOT PREPARATION
3811.02 BOOL  ; ROBOT FIXED POSITION PULSE
3811.03 BOOL  ; ROBOT FIXED POSITION PULSE 1 SCAN KEEP
3811.04 BOOL  ; ROBOT FIXED POSITION
3811.08 BOOL  ; ROBOT FAULT CLEAR TIMING
3811.09 BOOL  ; COMPLETION OF ROBOT FAULT CLEAR
3811.10 BOOL  ; Robot abnormal code reading
3811.11 BOOL  ; COMMAND PROCESSING COMPLETION
3811.12 BOOL  ; Robot abnormal code reading reset
3812.00 BOOL  ; AUTO RUNNING STOP PULSE
3812.01 BOOL  ; The robot doesn't stop
3812.02 BOOL  ; 1 CYCLE RUNNING STOP PULSE
3900.00 BOOL  ; LANGUAGE CHANGE ENGLISH
3900.01 BOOL  ; LANGUAGE CHANGE JAPANESE
4000.01 BOOL  ; Reference address reading beginning
4000.02 BOOL  ; It is reading it
4000.03 BOOL  ; Trigger
4000.04 BOOL  ; Reference address reading completion
4000.10 BOOL  ; Reading start
4000.11 BOOL  ; ID is being read
4000.12 BOOL  ; Trigger
4000.13 BOOL  ; Continuance
4000.14 BOOL  ; Completion
4000.15 BOOL  ; Reading completion
4001.00 BOOL  ; Reference address reading beginning
4001.01 BOOL  ; It is reading it
4001.02 BOOL  ; ﾄﾘｶﾞ
4001.03 BOOL  ; Reference address reading completion (Exchange unit of lane 1)
4002.08 BOOL  ; Writing start
4002.09 BOOL  ; ID is being written
4002.10 BOOL  ; Trigger
4002.11 BOOL  ; Continuance
4002.12 BOOL  ; Completion
4002.13 BOOL  ; Writing completion (Exchange unit of lane 1)
4004.01 BOOL  ; Reference address reading beginning
4004.02 BOOL  ; It is reading it
4004.03 BOOL  ; Trigger
4004.04 BOOL  ; Reference address reading completion
4004.09 BOOL  ; Fraction workpiece container
4004.10 BOOL  ; Reading start
4004.11 BOOL  ; ID is being read
4004.12 BOOL  ; Trigger
4004.13 BOOL  ; Continuance
4004.14 BOOL  ; Completion
4004.15 BOOL  ; Reading completion (Befor exchange unit of lane 1)
4005.00 BOOL  ; Reference address reading beginning
4005.01 BOOL  ; It is reading it
4005.02 BOOL  ; ﾄﾘｶﾞ
4005.03 BOOL  ; Reference address reading completion
4006.08 BOOL  ; Writing start
4006.09 BOOL  ; ID is being written
4006.10 BOOL  ; Trigger
4006.11 BOOL  ; Continuance
4006.12 BOOL  ; Completion
4006.13 BOOL  ; Writing completion (Befor exchange unit of lane 1)
4008.01 BOOL  ; Reference address reading beginning
4008.02 BOOL  ; It is reading it
4008.03 BOOL  ; Trigger
4008.04 BOOL  ; Reference address reading completion
4008.10 BOOL  ; Reading start
4008.11 BOOL  ; ID is being read
4008.12 BOOL  ; Trigger
4008.13 BOOL  ; Continuance
4008.14 BOOL  ; Completion
4008.15 BOOL  ; Reading completion (Exchange unit of lane 2)
4009.00 BOOL  ; Reference address reading beginning
4009.01 BOOL  ; It is reading it
4009.02 BOOL  ; Trigger
4009.03 BOOL  ; Reference address reading completion
4010.08 BOOL  ; Writing start
4010.09 BOOL  ; ID is being written
4010.10 BOOL  ; Trigger
4010.11 BOOL  ; Continuance
4010.12 BOOL  ; Completion
4010.13 BOOL  ; Writing completion (Exchange unit of lane 2)
4012.01 BOOL  ; Reference address reading beginning
4012.02 BOOL  ; It is reading it
4012.03 BOOL  ; Trigger
4012.04 BOOL  ; Reference address reading completion
4012.09 BOOL  ; Fraction workpiece container
4012.10 BOOL  ; Reading start
4012.11 BOOL  ; ID is being read
4012.12 BOOL  ; Trigger
4012.13 BOOL  ; Continuance
4012.14 BOOL  ; Completion
4012.15 BOOL  ; Reading completion (Befor exchange unit of lane 2)
4013.00 BOOL  ; Reference address reading beginning
4013.01 BOOL  ; It is reading it
4013.02 BOOL  ; ﾄﾘｶﾞ
4013.03 BOOL  ; Reference address reading completion
4014.08 BOOL  ; Writing start
4014.09 BOOL  ; ID is being written
4014.10 BOOL  ; Trigger
4014.11 BOOL  ; Continuance
4014.12 BOOL  ; Completion
4014.13 BOOL  ; Writing completion (Befor exchange unit of lane 2)
4101.12 BOOL  ; Data delivery completion signal
4101.13 BOOL  ; Completed receiving work information to the previous process
4102.03 BOOL  ; 01ST_NO INTERFERENCE
4103.00 BOOL  ; 01ST_1CY START PB on
4103.01 BOOL  ; 01ST_1CY RUN
4103.02 BOOL  ; 01ST_INDIV STEP START
4103.03 BOOL  ; 01ST_UNIT HOME POSITION PB
4103.04 BOOL  ; 01ST_UNIT HOME POSITION PB PLUSE
4104.00 BOOL  ; 01ST_CONDITION OF START(AUTO)
4104.01 BOOL  ; 01ST_CONDITION OF START(INDIV)
4104.04 BOOL  ; 01ST_CONDITION OF CYCLE START
4104.08 BOOL  ; 01ST_START RESET
4104.09 BOOL  ; 01ST_STEP UP ENABLE
4105.00 BOOL  ; 01ST_CYCLE RUNNING
4105.01 BOOL  ; 01ST_CYCLE RUNNING PLUSE
4105.02 BOOL  ; 01ST_STEP UP ENABLE
4105.15 BOOL  ; 01ST_CYCLE COMPLETE
4130.00 BOOL  ; 投入ﾊﾟﾚｯﾄｼﾌﾄ前進
4130.01 BOOL  ; 投入ﾊﾟﾚｯﾄｼﾌﾄ後退
4130.04 BOOL  ; 投入ﾊﾟﾚｯﾄ払出し前進
4130.05 BOOL  ; 投入ﾊﾟﾚｯﾄ払出し後退
4140.00 BOOL  ; LOADING CONVEYOR PALLET SHIFT FORWARD
4140.01 BOOL  ; LOADING CONVEYOR PALLET SHIFT BACKWARD
4140.04 BOOL  ; LOADING CONVEYOR PALLET DISCHARGE FORWARD
4140.05 BOOL  ; LOADING CONVEYOR PALLET DISCHARGE BACKWARD
4145.00 BOOL  ; 01ST_HOME POSITION
4145.01 BOOL  ; 01ST_CYCLE RUNNING
4152.00 BOOL  ; TRANSFER CARRIER NO INTERFERENCE
4152.10 BOOL  ; Fraction workpiece exhaust
4153.00 BOOL  ; 02ST_1CY START PB on
4153.01 BOOL  ; 02ST_1CY RUN
4153.02 BOOL  ; 02ST_INDIV STEP START
4153.03 BOOL  ; 02ST_UNIT HOME POSITION PB
4153.04 BOOL  ; 02ST_UNIT HOME POSITION PB PLUSE
4153.05 BOOL  ; 02ST_1CY START PB on PLUSE
4154.00 BOOL  ; 02ST_CONDITION OF START(AUTO)
4154.01 BOOL  ; 02ST_CONDITION OF START(INDIV)
4154.04 BOOL  ; 02ST_CONDITION OF CYCLE START
4154.08 BOOL  ; 02ST_START RESET
4154.09 BOOL  ; 02ST_STEP UP ENABLE
4155.00 BOOL  ; 02ST_CYCLE RUNNING
4155.01 BOOL  ; 02ST_CYCLE RUNNING PLUSE
4155.02 BOOL  ; 02ST_STEP UP ENABLE
4155.10 BOOL  ; CHUCK MISS OF LOADING WORKPIECE
4155.15 BOOL  ; 02ST_CYCLE COMPLETE
4180.00 BOOL  ; LOADER FORWARD
4180.01 BOOL  ; LOADER BACKWARD
4180.02 BOOL  ; LOADER DOWNWARD
4180.03 BOOL  ; LOADER UPWARD
4180.04 BOOL  ; TURN LOADER CHUCK TURN
4180.05 BOOL  ; TURN LOADER RECHUCK TURN
4180.06 BOOL  ; LOADER CHUCK CLAMP
4180.07 BOOL  ; LOADER CHUCK UNCLAMP
4190.00 BOOL  ; LOADER FORWARD
4190.01 BOOL  ; LOADER BACKWARD
4190.02 BOOL  ; LOADER DOWNWARD
4190.03 BOOL  ; LOADER UPWARD
4190.04 BOOL  ; TURN LOADER CHUCK TURN
4190.05 BOOL  ; TURN LOADER RECHUCK TURN
4190.06 BOOL  ; LOADER CHUCK CLAMP
4190.07 BOOL  ; LOADER CHUCK UNCLAMP
4195.00 BOOL  ; 02ST_HOME POSITION
4195.01 BOOL  ; 02ST_CYCLE RUNNING
4202.00 BOOL  ; Workpiece clamp downward receipt completion
4202.01 BOOL  ; Measurement start receipt completion
4202.02 BOOL  ; Transfer-carrier backward permission signal
4202.03 BOOL  ; Measurement completion signal
4202.04 BOOL  ; Workpiece clamp upward receipt completion
4202.06 BOOL  ; TRANSFER CARRIER LIFT UPWARD
4202.07 BOOL  ; TRANSFER CARRIER LIFT DOWNWARD
4202.08 BOOL  ; SUB TRANSFER CARRIER LIFT UPWARD
4202.09 BOOL  ; SUB TRANSFER CARRIER LIFT DOWNWARD
4202.10 BOOL  ; All Station Process Complete
4203.00 BOOL  ; 03ST_1CY START PB on
4203.01 BOOL  ; 03ST_1CY RUN
4203.02 BOOL  ; 03ST_INDIV STEP START
4203.03 BOOL  ; 03ST_UNIT HOME POSITION PB
4203.04 BOOL  ; 03ST_UNIT HOME POSITION PB PLUSE
4204.00 BOOL  ; 03ST_CONDITION OF START(AUTO)
4204.01 BOOL  ; 03ST_CONDITION OF START(INDIV)
4204.04 BOOL  ; 03ST_CONDITION OF CYCLE START
4204.08 BOOL  ; 03ST_START RESET
4204.09 BOOL  ; 03ST_STEP UP ENABLE
4205.00 BOOL  ; 03ST_CYCLE RUNNING
4205.01 BOOL  ; 03ST_CYCLE RUNNING PLUSE
4205.02 BOOL  ; 03ST_STEP UP ENABLE
4205.15 BOOL  ; 03ST_CYCLE COMPLETE
4220.00 BOOL  ; TRANSFER CARRIER FORWARD END
4220.01 BOOL  ; TRANSFER CARRIER FORWARD
4220.02 BOOL  ; Completion storage clearness
4230.00 BOOL  ; TRANSFER CARRIER LIFT UPWARD
4230.01 BOOL  ; TRANSFER CARRIER LIFT DOWNWARD
4230.02 BOOL  ; TRANSFER CARRIER FORWARD
4230.03 BOOL  ; TRANSFER CARRIER BACKWARD
4230.04 BOOL  ; SUB TRANSFER CARRIER LIFT UPWARD
4230.05 BOOL  ; SUB TRANSFER CARRIER LIFT DOWNWARD
4230.06 BOOL  ; Workpiece Clamp Down
4230.07 BOOL  ; Workpiece Clamp Up
4240.00 BOOL  ; TRANSFER CARRIER LIFT UPWARD
4240.01 BOOL  ; TRANSFER CARRIER LIFT DOWNWARD
4240.02 BOOL  ; TRANSFER CARRIER FORWARD
4240.03 BOOL  ; TRANSFER CARRIER BACKWARD
4240.08 BOOL  ; TRANSFER CARRIER NO INTERFERENCE
4243.00 BOOL  ; Workpiece clamp downward signal
4243.01 BOOL  ; Measurement strating signal
4243.02 BOOL  ; Transfer-carrier backward signal receipt
4243.03 BOOL  ; Measurement completion receipt
4243.04 BOOL  ; Workpiece clamp upward signal
4243.06 BOOL  ; TRANSFER CARRIER NO INTERFERENCE
4243.07 BOOL  ; WorkPiece Ready For Measuring Impulse and Resistance
4243.10 BOOL  ; TRANSFER CARRIER FORWARD
4245.00 BOOL  ; 03ST_HOME POSITION
4245.01 BOOL  ; 03ST_CYCLE RUNNING
4245.04 BOOL  ; Lifter rising edge
4253.00 BOOL  ; 04ST_1CY START PB on
4253.01 BOOL  ; 04ST_1CY RUN
4253.02 BOOL  ; 04ST_INDIV STEP START
4253.03 BOOL  ; 04ST_UNIT HOME POSITION PB
4253.04 BOOL  ; 04ST_UNIT HOME POSITION PB PLUSE
4254.00 BOOL  ; 04ST_CONDITION OF START(AUTO)
4254.01 BOOL  ; 04ST_CONDITION OF START(INDIV)
4254.04 BOOL  ; 04ST_CONDITION OF CYCLE START
4254.08 BOOL  ; 04ST_START RESET
4254.09 BOOL  ; 04ST_STEP UP ENABLE
4255.00 BOOL  ; 04ST_CYCLE RUNNING
4255.01 BOOL  ; 04ST_CYCLE RUNNING PLUSE
4255.02 BOOL  ; 04ST_STEP UP ENABLE
4255.10 BOOL  ; THICKNESS OF CORE L
4255.11 BOOL  ; THICKNESS OF CORE S
4255.12 BOOL  ; DEFECT OF THICKNESS OF CORE
4255.15 BOOL  ; 04ST_CYCLE COMPLETE
4280.00 BOOL  ; WORKPIECE PUSHER FORWARD
4290.00 BOOL  ; WORKPIECE PUSHER FORWARD
4290.04 BOOL  ; Start of distinction of thickness in core
4295.00 BOOL  ; 04ST_HOME POSITION
4295.01 BOOL  ; 04ST_CYCLE RUNNING
4302.01 BOOL  ; Measurement strating signal
4302.03 BOOL  ; Measurement completion receipt
4302.06 BOOL  ; TRANSFER CARRIER NO INTERFERENCE
4303.00 BOOL  ; 05ST_1CY START PB on
4303.01 BOOL  ; 05ST_1CY RUN
4303.02 BOOL  ; 05ST_INDIV STEP START
4303.03 BOOL  ; 05ST_UNIT HOME POSITION PB
4303.04 BOOL  ; 05ST_UNIT HOME POSITION PB PLUSE
4304.00 BOOL  ; 05ST_CONDITION OF START(AUTO)
4304.01 BOOL  ; 05ST_CONDITION OF START(INDIV)
4304.04 BOOL  ; 05ST_CONDITION OF CYCLE START
4304.08 BOOL  ; 05ST_START RESET
4304.09 BOOL  ; 05ST_STEP UP ENABLE
4305.00 BOOL  ; 05ST_CYCLE RUNNING
4305.01 BOOL  ; 05ST_CYCLE RUNNING PLUSE
4305.02 BOOL  ; 05ST_STEP UP ENABLE
4305.15 BOOL  ; 05ST_CYCLE COMPLETE
4313.00 BOOL  ; WITHSTAND VOLTAGE TESTER RESET
4313.01 BOOL  ; WITHSTAND VOLTAGE TESTER READY
4330.04 BOOL  ; WITHSTAND VOLTAGE TEST START
4334.00 BOOL  ; INSULATION  TEST START
4334.01 BOOL  ; INSULATION  TEST START PULSE
4334.02 BOOL  ; Contact inspection relay ON
4334.03 BOOL  ; Contact inspection start
4334.04 BOOL  ; Contact OK
4334.05 BOOL  ; Contact NG
4334.06 BOOL  ; Circuit connection
4334.07 BOOL  ; RESET
4334.08 BOOL  ; START CONDITION
4334.09 BOOL  ; INSULATION TEST
4334.10 BOOL  ; INSULATION OK
4334.11 BOOL  ; INSULATION NG
4334.13 BOOL  ; INSULATION TEST COMPLETE
4335.07 BOOL  ; INSULATION CYCLE END
4335.10 BOOL  ; Repeated challenge
4340.00 BOOL  ; TRANSFER CARRIER LIFT UPWARD
4340.01 BOOL  ; TRANSFER CARRIER LIFT DOWNWARD
4340.04 BOOL  ; INSULATION  TEST START
4343.01 BOOL  ; Measurement strating signal
4343.03 BOOL  ; Measurement completion receipt
4343.06 BOOL  ; TRANSFER CARRIER LIFT UPWARD
4343.07 BOOL  ; TRANSFER CARRIER LIFT DOWNWARD
4345.00 BOOL  ; 05ST_HOME POSITION
4345.01 BOOL  ; 05ST_CYCLE RUNNING
4352.01 BOOL  ; Measurement strating signal
4352.02 BOOL  ; XXXXXX
4352.03 BOOL  ; Measurement completion receipt
4352.06 BOOL  ; TRANSFER CARRIER NO INTERFERENCE
4353.00 BOOL  ; 06ST_1CY START PB on
4353.01 BOOL  ; 06ST_1CY RUN
4353.02 BOOL  ; 06ST_INDIV STEP START
4353.03 BOOL  ; 06ST_UNIT HOME POSITION PB
4353.04 BOOL  ; 06ST_UNIT HOME POSITION PB PLUSE
4354.00 BOOL  ; 06ST_CONDITION OF START(AUTO)
4354.01 BOOL  ; 06ST_CONDITION OF START(INDIV)
4354.04 BOOL  ; 06ST_CONDITION OF CYCLE START
4354.08 BOOL  ; 06ST_START RESET
4354.09 BOOL  ; 06ST_STEP UP ENABLE
4355.00 BOOL  ; 06ST_CYCLE RUNNING
4355.01 BOOL  ; 06ST_CYCLE RUNNING PLUSE
4355.02 BOOL  ; 06ST_STEP UP ENABLE
4355.15 BOOL  ; 06ST_CYCLE COMPLETE
4380.02 BOOL  ; POSITIONING ARROW FORWARD
4380.06 BOOL  ; WORKPIECE DRIVE HIGH SPEED
4380.07 BOOL  ; WORKPIECE DRIVE MIDDLE SPEED
4380.10 BOOL  ; COUNT STOP
4380.11 BOOL  ; COUNT RESET
4380.12 BOOL  ; Measurement start
4380.13 BOOL  ; Measurement stop
4382.00 BOOL  ; SWING OK (SHAFT END)
4382.01 BOOL  ; SWING NG (SHAFT END)
4382.02 BOOL  ; SWING OK (WORM)
4382.03 BOOL  ; SWING NG (WORM)
4382.04 BOOL  ; SWING OK
4382.05 BOOL  ; SWING NG
4382.06 BOOL  ; COIL END L
4382.07 BOOL  ; COIL END S
4382.08 BOOL  ; OIL END NG
4382.11 BOOL  ; DISTINCTION START OF COIL END
4382.12 BOOL  ; WORKPIECE OF COIL END L
4390.00 BOOL  ; TRANSFER CARRIER LIFT UPWARD
4390.01 BOOL  ; TRANSFER CARRIER LIFT DOWNWARD
4390.02 BOOL  ; POSITIONING ARROW FORWARD
4390.03 BOOL  ; POSITIONING ARROW BACKWARD
4390.04 BOOL  ; POSITIONING START
4390.08 BOOL  ; SWING MEASURE START
4393.01 BOOL  ; Measurement strating signal
4393.03 BOOL  ; Measurement completion receipt
4393.06 BOOL  ; TRANSFER CARRIER LIFT UPWARD
4393.07 BOOL  ; TRANSFER CARRIER LIFT DOWNWARD
4395.00 BOOL  ; 06ST_HOME POSITION
4395.01 BOOL  ; 06ST_CYCLE RUNNING
4402.00 BOOL  ; Workpiece clamp downward signal
4402.01 BOOL  ; Measurement strating signal
4402.02 BOOL  ; Transfer-carrier backward signal receipt
4402.03 BOOL  ; Measurement completion receipt
4402.04 BOOL  ; Workpiece clamp upward signal
4402.06 BOOL  ; TRANSFER CARRIER NO INTERFERENCE
4402.08 BOOL  ; WORKPIECE CLAMP DOWNWARD
4402.09 BOOL  ; WORKPIECE CLAMP UPWARD
4402.10 BOOL  ; ｲﾝﾊﾟﾙｽST測定ﾜｰｸ無し
4402.13 BOOL  ; WorkPisece Ready For Measuring
4403.00 BOOL  ; 07ST_1CY START PB on
4403.01 BOOL  ; 07ST_1CY RUN
4403.02 BOOL  ; 07ST_INDIV STEP START
4403.03 BOOL  ; 07ST_UNIT HOME POSITION PB
4403.04 BOOL  ; 07ST_UNIT HOME POSITION PB PLUSE
4404.00 BOOL  ; 07ST_CONDITION OF START(AUTO)
4404.01 BOOL  ; 07ST_CONDITION OF START(INDIV)
4404.04 BOOL  ; 07ST_CONDITION OF CYCLE START
4404.08 BOOL  ; 07ST_START RESET
4404.09 BOOL  ; 07ST_STEP UP ENABLE
4405.00 BOOL  ; 07ST_CYCLE RUNNING
4405.01 BOOL  ; 07ST_CYCLE RUNNING PLUSE
4405.02 BOOL  ; 07ST_STEP UP ENABLE
4405.03 BOOL  ; Resistance measurement unit_preceding operation
4405.15 BOOL  ; 07ST_CYCLE COMPLETE
4420 CHANNEL  ; PAIR RESISTANCE FREQUENCY
4420.01 BOOL  ; PAIR RESISTANCE FREQUENCY *1
4420.02 BOOL  ; PAIR RESISTANCE FREQUENCY *2
4420.03 BOOL  ; PAIR RESISTANCE FREQUENCY *3
4420.04 BOOL  ; PAIR RESISTANCE FREQUENCY *4
4420.05 BOOL  ; PAIR RESISTANCE FREQUENCY *5
4420.06 BOOL  ; PAIR RESISTANCE FREQUENCY *6
4420.07 BOOL  ; Number of counter electrode resistance * 7
4420.08 BOOL  ; Number of counter electrode resistance * 8
4420.09 BOOL  ; Number of counter electrode resistance * 9
4421 CHANNEL  ; Counter electrode resistance Current measurement count (180 °)
4421.01 BOOL  ; Number of counter electrode resistance 1 *
4421.02 BOOL  ; Number of adjacent resistances * 2
4421.03 BOOL  ; Number of adjacent resistances * 3
4421.04 BOOL  ; Number of adjacent resistances * 4
4421.05 BOOL  ; Number of adjacent resistances * 5
4421.06 BOOL  ; Number of adjacent resistances * 6
4421.07 BOOL  ; Number of adjacent resistances * 7
4421.08 BOOL  ; Number of adjacent resistances * 8
4421.09 BOOL  ; Number of adjacent resistances * 9
4430.02 BOOL  ; WORKPIECE CLAMP DOWNWARD
4430.03 BOOL  ; WORKPIECE CLAMP UPWARD
4430.07 BOOL  ; Resistance probe advance completed
4430.08 BOOL  ; Resistance probe retreat confirmation
4430.09 BOOL  ; Resistance probe retreat_for investigation
4430.10 BOOL  ; CONTACT PROBE IN RESISTANCE FORWARD
4430.14 BOOL  ; Start resistance measurement (80 ° counter electrode)
4431.01 BOOL  ; NUMBER OF TURNS CHECK START
4431.02 BOOL  ; NUMBER OF TURNS CHECK RUNNING
4431.03 BOOL  ; $?St$Bk?_#[14] / NUMBER OF TURNS CHECK "TRIG"$?St$Bk?_#[14]
4431.04 BOOL  ; NUMBER OF TURNS RESULT CONFIRMATION
4431.05 BOOL  ; $?St$Bk?_#[15] / NUMBER OF TURNS CHECK "H"$?St$Bk?_#[15]
4431.06 BOOL  ; $?St$Bk?_#[16] / NUMBER OF TURNS CHECK "L"$?St$Bk?_#[16]
4431.07 BOOL  ; $?St$Bk?_#[17] / NUMBER OF TURNS CHECK "NG"$?St$Bk?_#[17]
4431.08 BOOL  ; ﾀｰﾝ数判別ﾘﾚｰ切替
4431.14 BOOL  ; Start resistance measurement (180 ° counter electrode)
4432.03 BOOL  ; Counter electrode resistance measurement start (80 °)
4432.04 BOOL  ; PAIR BCD OUTPUT STABILITY
4432.05 BOOL  ; Resistance stability output
4432.06 BOOL  ; Measurement end OFF memory
4432.07 BOOL  ; Adjacent resistance measurement end pulse
4432.08 BOOL  ; PAIR RESISTANCE MEASUREMENT
4432.09 BOOL  ; Reached the number of counter electrode measurements (80 °)
4432.10 BOOL  ; PAIR RESISTANCE MEASUREMENT COMPLETE
4432.11 BOOL  ; Counter electrode resistance OK Next (80 °)
4432.15 BOOL  ; Measurement end OFF
4433.00 BOOL  ; XXXXXX
4433.03 BOOL  ; Counter electrode resistance measurement start (180 °)
4433.04 BOOL  ; Counterpole BCD output stable (180 °)
4433.06 BOOL  ; Adjacent measurement end OFF memory
4433.08 BOOL  ; Counter electrode resistance measurement (180 °)
4433.09 BOOL  ; PAIR RESISTANCE OK
4433.10 BOOL  ; 180 Degree  RESISTANCE Complete
4433.11 BOOL  ; Counter electrode resistance OK Pair (180 °)
4434.00 BOOL  ; PAIR RESISTANCE OK
4434.01 BOOL  ; PAIR RESISTANCE NG
4434.02 BOOL  ; 180 ° counter electrode contact resistance OK
4434.03 BOOL  ; 180 ° counter electrode contact resistance NG
4434.09 BOOL  ; Resistor retry start
4434.10 BOOL  ; There is NG
4434.11 BOOL  ; RESET PULSE OF RESTART
4434.12 BOOL  ; Retry Operation
4435.00 BOOL  ; RESISTANCE OK
4435.01 BOOL  ; RESISTANCE NG
4435.02 BOOL  ; Resistance NG ( For Retry)
4435.03 BOOL  ; Resistance NG (180 °)
4436.01 BOOL  ; Code No.1(resistance)
4436.02 BOOL  ; Code No.2(resistance)
4436.03 BOOL  ; Code No.3(resistance)
4436.04 BOOL  ; PAIR RESISTANCE OK (80 Degree)
4436.05 BOOL  ; PAIR RESISTANCE NG ( 80 Degree)
4436.06 BOOL  ; Next RESISTANCE OK (180 Degree)
4436.07 BOOL  ; Next RESISTANCE NG (180 Degree)
4436.08 BOOL  ; Code No.8(resistance)
4436.09 BOOL  ; Code No.9(resistance)
4436.15 BOOL  ; Code No. distinction
4437.01 BOOL  ; Code No.1 (resistance) selection
4437.02 BOOL  ; Code No.2 (resistance) selection
4437.03 BOOL  ; Code No.3 (resistance) selection
4437.04 BOOL  ; Code No.4 (resistance) selection
4437.05 BOOL  ; Code No.5 (resistance) selection
4437.06 BOOL  ; Code No.6 (resistance) selection
4437.07 BOOL  ; Code No.7 (resistance) selection
4437.08 BOOL  ; Code No.8 (resistance) selection
4437.09 BOOL  ; Code No.9 (resistance) selection
4438 CHANNEL  ; CODE No.
4438.01 BOOL  ; Code No.1 selection
4438.02 BOOL  ; Code No.2 selection
4438.03 BOOL  ; Code No.3 selection
4438.04 BOOL  ; Code No.4 selection
4438.05 BOOL  ; Code No.5 selection
4438.06 BOOL  ; Code No.6 selection
4438.07 BOOL  ; Code No.7 selection
4438.08 BOOL  ; Code No.8 selection
4438.09 BOOL  ; Code No.9 selection
4439.00 BOOL  ; Contact Probe Upper Resistance Forward
4439.01 BOOL  ; Contact Probe Lower Resistance Forward
4439.02 BOOL  ; COIL END L
4439.03 BOOL  ; COIL END S
4439.04 BOOL  ; Product number distinction OK
4439.05 BOOL  ; Product number distinction NG
4439.06 BOOL  ; Product number data transfer
4440.02 BOOL  ; WORKPIECE CLAMP DOWNWARD
4440.03 BOOL  ; WORKPIECE CLAMP UPWARD
4440.06 BOOL  ; TRANSFER CARRIER LIFT UPWARD
4440.07 BOOL  ; TRANSFER CARRIER LIFT DOWNWARD
4440.10 BOOL  ; CONTACT PROBE IN RESISTANCE FORWARD
4440.14 BOOL  ; RESISTANCE MEASUREMENT START
4443.00 BOOL  ; Workpiece clamp downward signal
4443.01 BOOL  ; Measurement strating signal
4443.02 BOOL  ; Transfer-carrier backward signal receipt
4443.03 BOOL  ; Measurement completion receipt
4443.04 BOOL  ; Workpiece clamp upward signal
4443.06 BOOL  ; TRANSFER CARRIER LIFT UPWARD
4443.07 BOOL  ; TRANSFER CARRIER LIFT DOWNWARD
4444.08 BOOL  ; RESISTANCE MEASURED VALUE LOWER CAPTURE COMPL
4444.09 BOOL  ; 1X Measure Judgment
4444.10 BOOL  ; 1x Judgment Good
4444.11 BOOL  ; RESISTANCE VALUE READING MONITOR
4444.13 BOOL  ; 1x Judgment Good
4444.14 BOOL  ; 1x Judgment No Good
4445.00 BOOL  ; 07ST_HOME POSITION
4445.01 BOOL  ; 07ST_CYCLE RUNNING
4452.00 BOOL  ; Workpiece clamp downward signal
4452.01 BOOL  ; Measurement strating signal
4452.02 BOOL  ; Transfer-carrier backward signal receipt
4452.03 BOOL  ; Measurement completion receipt
4452.04 BOOL  ; Workpiece clamp upward signal
4452.06 BOOL  ; TRANSFER CARRIER NO INTERFERENCE
4453.00 BOOL  ; 08ST_1CY START PB on
4453.01 BOOL  ; 08ST_1CY RUN
4453.02 BOOL  ; 08ST_INDIV STEP START
4453.03 BOOL  ; 08ST_UNIT HOME POSITION PB
4453.04 BOOL  ; 08ST_UNIT HOME POSITION PB PLUSE
4454.00 BOOL  ; 08ST_CONDITION OF START(AUTO)
4454.01 BOOL  ; 08ST_CONDITION OF START(INDIV)
4454.04 BOOL  ; 08ST_CONDITION OF CYCLE START
4454.08 BOOL  ; 08ST_START RESET
4454.09 BOOL  ; 08ST_STEP UP ENABLE
4455.00 BOOL  ; 08ST_CYCLE RUNNING
4455.01 BOOL  ; 08ST_CYCLE RUNNING PLUSE
4455.02 BOOL  ; 08ST_STEP UP ENABLE
4455.03 BOOL  ; Impression measurement unit_preceding operation
4455.15 BOOL  ; 08ST_CYCLE COMPLETE
4456.00 BOOL  ; CONTACT PROBE IN INPULSE BACKWARD
4457.00 BOOL  ; Lower impulse probe forward end holding
4457.01 BOOL  ; Upper impulse probe forward end holding
4480.00 BOOL  ; WORKPIECE CLAMP DOWNWARD
4480.01 BOOL  ; WORKPIECE CLAMP UPWARD
4480.02 BOOL  ; CONTACT PROBE IN INPULSE FORWARD
4481.06 BOOL  ; PAIR IMPULSE MEASUREMENT START
4481.07 BOOL  ; NEXT IMPULSE MEASUREMENT START
4481.08 BOOL  ; Trigger signal
4481.09 BOOL  ; During counter electrode measurement
4481.11 BOOL  ; 隣接測定開始（解析用）
4482.04 BOOL  ; PAIR PAGE SET
4482.05 BOOL  ; The first relay switch
4482.06 BOOL  ; Completion once
4482.07 BOOL  ; PAIR POLE NG
4482.09 BOOL  ; PAIR POLE OK
4484.04 BOOL  ; NEXT PAGE SET
4484.05 BOOL  ; Adjacent page SET
4484.06 BOOL  ; Completion once
4484.07 BOOL  ; NEXT POLE NG
4484.09 BOOL  ; NEXT POLE  OK
4484.10 BOOL  ; Judgment completion of impulse
4484.12 BOOL  ; NG COUNT 1 PULSE
4484.14 BOOL  ; RESET
4486.00 BOOL  ; There is NG
4490.00 BOOL  ; WORKPIECE CLAMP DOWNWARD
4490.01 BOOL  ; WORKPIECE CLAMP UPWARD
4490.02 BOOL  ; CONTACT PROBE IN INPULSE FORWARD
4490.04 BOOL  ; TRANSFER CARRIER LIFT UPWARD
4490.05 BOOL  ; TRANSFER CARRIER LIFT DOWNWARD
4490.06 BOOL  ; IMPULSE MEASUREMENT START
4490.08 BOOL  ; PAIR RERAY PULSE
4490.09 BOOL  ; NEXT RERAY PULSE
4490.10 BOOL  ; Relay ON to pair pole
4490.11 BOOL  ; Relay ON to next pole
4490.12 BOOL  ; Step mode ON pulse
4490.13 BOOL  ; Step mode start
4490.14 BOOL  ; Step mode ON
4490.15 BOOL  ; WABE INDICATE ON PULSE
4491.05 BOOL  ; 対極測定開始
4491.06 BOOL  ; PAIR IMPULSE MEASURE
4491.07 BOOL  ; One time end
4491.11 BOOL  ; NEXT IMPULSE MEASUREMENT START PULSE
4491.12 BOOL  ; PAIR IMPULSE MEASUREMENT START
4491.13 BOOL  ; PAIR IMPULSE MEASUREMENT COMPLETE
4491.15 BOOL  ; STEP UP
4492.04 BOOL  ; 隣接測定開始
4492.05 BOOL  ; NEXT IMPULSE MEASUREMENT START
4492.06 BOOL  ; NEXT IMPULSE MEASURE
4492.07 BOOL  ; One time end
4492.12 BOOL  ; NEXT IMPULSE MEASUREMENT START
4492.13 BOOL  ; IMPULSE MEASUREMENT COMPLETE
4492.15 BOOL  ; STEP UP
4493.00 BOOL  ; Workpiece clamp downward signal
4493.01 BOOL  ; Measurement strating signal
4493.02 BOOL  ; Transfer-carrier backward signal receipt
4493.03 BOOL  ; Measurement completion receipt
4493.04 BOOL  ; Workpiece clamp upward signal
4493.06 BOOL  ; TRANSFER CARRIER LIFT UPWARD
4493.07 BOOL  ; TRANSFER CARRIER LIFT DOWNWARD
4493.08 BOOL  ; WORKPIECE CLAMP DOWNWARD
4493.09 BOOL  ; WORKPIECE CLAMP UPWARD
4495.00 BOOL  ; 08ST_HOME POSITION
4495.01 BOOL  ; 08ST_CYCLE RUNNING
4502.01 BOOL  ; Insert starting signal
4502.03 BOOL  ; Insert completion receipt
4502.06 BOOL  ; TRANSFER CARRIER NO INTERFERENCE
4502.07 BOOL  ; WorkPiece Clamp Down
4502.08 BOOL  ; Workpiecee Clamp Up
4503.00 BOOL  ; 09ST_1CY START PB on
4503.01 BOOL  ; 09ST_1CY RUN
4503.02 BOOL  ; 09ST_INDIV STEP START
4503.03 BOOL  ; 09ST_UNIT HOME POSITION PB
4503.04 BOOL  ; 09ST_UNIT HOME POSITION PB PLUSE
4504.00 BOOL  ; 09ST_CONDITION OF START(AUTO)
4504.01 BOOL  ; 09ST_CONDITION OF START(INDIV)
4504.04 BOOL  ; 09ST_CONDITION OF CYCLE START
4504.08 BOOL  ; 09ST_START RESET
4504.09 BOOL  ; 09ST_STEP UP ENABLE
4505.00 BOOL  ; 09ST_CYCLE RUNNING
4505.01 BOOL  ; 09ST_CYCLE RUNNING PLUSE
4505.02 BOOL  ; 09ST_STEP UP ENABLE
4505.06 BOOL  ; Bearing inside and outside check OK
4505.07 BOOL  ; Bearing inside and outside check NG
4505.15 BOOL  ; 09ST_CYCLE COMPLETE
4530.02 BOOL  ; BEARING INSERT (HIGH SPEED) FORWARD
4530.03 BOOL  ; BEARING INSERT (HIGH SPEED) BACKWARD
4530.04 BOOL  ; BEARING INSERT (HIGH PRESSURE) ON
4530.05 BOOL  ; BEARING INSERT (HIGH PRESSURE) OFF
4530.06 BOOL  ; BEARING SHUTTER DOWNWARD
4530.07 BOOL  ; BEARING SHUTTER UPWARD
4530.08 BOOL  ; BEARING GUIDE FORWARD
4530.09 BOOL  ; BEARING GUIDE BACKWARD
4530.10 BOOL  ; BEARING ESCAPE FORWARD
4530.11 BOOL  ; BEARING ESCAPE BACKWARD
4530.12 BOOL  ; Work Clamp DownWard
4540.00 BOOL  ; SUB TRANSFER CARRIER LIFT UPWARD
4540.01 BOOL  ; SUB TRANSFER CARRIER LIFT DOWNWARD
4540.02 BOOL  ; BEARING INSERT (HIGH SPEED) FORWARD
4540.03 BOOL  ; BEARING INSERT (HIGH SPEED) BACKWARD
4540.04 BOOL  ; BEARING INSERT (HIGH PRESSURE) ON
4540.05 BOOL  ; BEARING INSERT (HIGH PRESSURE) OFF
4540.06 BOOL  ; BEARING SHUTTER DOWNWARD
4540.07 BOOL  ; BEARING SHUTTER UPWARD
4540.08 BOOL  ; BEARING GUIDE FORWARD
4540.09 BOOL  ; BEARING GUIDE BACKWARD
4540.10 BOOL  ; BEARING ESCAPE FORWARD
4540.11 BOOL  ; BEARING ESCAPE BACKWARD
4540.12 BOOL  ; Work Clamp DownWard
4540.13 BOOL  ; Work Clamp UpWard
4543.00 BOOL  ; WorkPiece Clamp Down Confirm
4543.01 BOOL  ; Insert start receipt completion
4543.03 BOOL  ; Insert completion signal
4543.08 BOOL  ; SUB TRANSFER CARRIER LIFT UPWARD
4543.09 BOOL  ; SUB TRANSFER CARRIER LIFT DOWNWARD
4543.10 BOOL  ; IND_Work Clamp DownWard
4543.11 BOOL  ; IND_Work Clamp UpWard
4545.00 BOOL  ; 09ST_HOME POSITION
4545.01 BOOL  ; 09ST_CYCLE RUNNING
4552.01 BOOL  ; Measurement strating signal
4552.03 BOOL  ; Measurement completion receipt
4552.04 BOOL  ; WORKPIECE CLAMP UPWARD
4552.05 BOOL  ; WORKPIECE CLAMP DOWNWARD
4552.06 BOOL  ; TRANSFER CARRIER NO INTERFERENCE
4553.00 BOOL  ; 10ST_1CY START PB on
4553.01 BOOL  ; 10ST_1CY RUN
4553.02 BOOL  ; 10ST_INDIV STEP START
4553.03 BOOL  ; 10ST_UNIT HOME POSITION PB
4553.04 BOOL  ; 10ST_UNIT HOME POSITION PB PLUSE
4554.00 BOOL  ; 10ST_CONDITION OF START(AUTO)
4554.01 BOOL  ; 10ST_CONDITION OF START(INDIV)
4554.04 BOOL  ; 10ST_CONDITION OF CYCLE START
4554.08 BOOL  ; 10ST_START RESET
4554.09 BOOL  ; 10ST_STEP UP ENABLE
4555.00 BOOL  ; 10ST_CYCLE RUNNING
4555.01 BOOL  ; 10ST_CYCLE RUNNING PLUSE
4555.02 BOOL  ; 10ST_STEP UP ENABLE
4555.15 BOOL  ; 10ST_CYCLE COMPLETE
4580.04 BOOL  ; LENGTH MEASUREMENT FORWARD
4580.05 BOOL  ; LENGTH MEASUREMENT BACKWARD
4580.06 BOOL  ; Work press rise from full length measurement
4580.12 BOOL  ; Confirmation of completion of preset
4580.14 BOOL  ; Full length measurement work hold down (automatic)
4580.15 BOOL  ; Work press rise from full length measurement (automatic)
4582.00 BOOL  ; OVERALL LENGTH OK
4582.01 BOOL  ; BEARING INSERT LENGTH OK
4582.02 BOOL  ; LENGTH CHECK OK
4582.03 BOOL  ; LENGTH CHECK NG
4590.00 BOOL  ; SUB TRANSFER CARRIER LIFT UPWARD
4590.01 BOOL  ; SUB TRANSFER CARRIER LIFT DOWNWARD
4590.04 BOOL  ; LENGTH MEASUREMENT FORWARD
4590.05 BOOL  ; LENGTH MEASUREMENT BACKWARD
4590.08 BOOL  ; LENGTH CHECK START
4590.09 BOOL  ; Work Clamp DownWard
4590.10 BOOL  ; Work Clamp UpWard
4591.00 BOOL  ; 0 MASTER SETTING
4591.01 BOOL  ; 0 MASTER SETTING PULSE
4591.04 BOOL  ; Upper limit master check
4591.05 BOOL  ; UPPER LIMIT MASTER SETTING PULSE
4591.06 BOOL  ; #NAME?
4591.08 BOOL  ; Lower limit master check
4591.09 BOOL  ; #NAME?
4591.10 BOOL  ; #NAME?
4592.00 BOOL  ; SUB TRANSFER CARRIER LIFT UPWARD
4592.01 BOOL  ; SUB TRANSFER CARRIER LIFT DOWNWARD
4592.04 BOOL  ; LENGTH MEASUREMENT FORWARD
4592.05 BOOL  ; LENGTH MEASUREMENT BACKWARD
4592.06 BOOL  ; High-speed counter opening gate
4592.07 BOOL  ; High-speed counter close gate
4592.08 BOOL  ; High-speed counter preset
4592.12 BOOL  ; Priset completion
4593.01 BOOL  ; Measurement strating signal
4593.03 BOOL  ; Measurement completion receipt
4593.08 BOOL  ; SUB TRANSFER CARRIER LIFT UPWARD
4593.09 BOOL  ; SUB TRANSFER CARRIER LIFT DOWNWARD
4593.10 BOOL  ; IND_Work Clamp DownWard
4593.11 BOOL  ; IND_Work Clamp UpWard
4595.00 BOOL  ; 10ST_HOME POSITION
4595.01 BOOL  ; 10ST_CYCLE RUNNING
4601.01 BOOL  ; Stacking container exhaust completion (Lane 1)
4601.02 BOOL  ; Stacking container exhaust completion (Lane 2)
4601.03 BOOL  ; 16ST_1CY RUN
4601.04 BOOL  ; 19ST_1CY RUN
4602.01 BOOL  ; TAKING-OUT SIGNAL OF WORKPIECE
4602.02 BOOL  ; Transfer-carrier backward signal receipt
4603.00 BOOL  ; 11ST_1CY START PB on
4603.01 BOOL  ; 11ST_1CY RUN
4603.02 BOOL  ; 11ST_INDIV STEP START
4603.03 BOOL  ; 11ST_UNIT HOME POSITION PB
4603.04 BOOL  ; 11ST_UNIT HOME POSITION PB PLUSE
4604.00 BOOL  ; 11ST_CONDITION OF START(AUTO)
4604.01 BOOL  ; 11ST_CONDITION OF START(INDIV)
4604.04 BOOL  ; 11ST_CONDITION OF CYCLE START
4604.08 BOOL  ; 11ST_START RESET
4604.09 BOOL  ; 11ST_STEP UP ENABLE
4605.00 BOOL  ; 11ST_CYCLE RUNNING
4605.01 BOOL  ; 11ST_CYCLE RUNNING PLUSE
4605.02 BOOL  ; 11ST_STEP UP ENABLE
4605.03 BOOL  ; Fraction workpiece exhaust start
4605.15 BOOL  ; 11ST_CYCLE COMPLETE
4620.00 BOOL  ; EXCHANGE CONTAINER (LANE 1)
4620.01 BOOL  ; EXCHANGE CONTAINER (LANE 2)
4620.02 BOOL  ; CONTAINER BEFOR EXCHANGE (LANE 1)
4620.03 BOOL  ; CONTAINER BEFOR EXCHANGE (LANE 2)
4621 CHANNEL  ; Flow product number (Lane 1)
4621.01 BOOL  ; Flow product number code No.1 (Lane 1)
4621.02 BOOL  ; Flow product number code No.2 (Lane 1)
4621.03 BOOL  ; Flow product number code No.3 (Lane 1)
4621.04 BOOL  ; Flow product number code No.4 (Lane 1)
4621.05 BOOL  ; Flow product number code No.5 (Lane 1)
4621.06 BOOL  ; Flow product number code No.6 (Lane 1)
4621.07 BOOL  ; Flow product number code No.7 (Lane 1)
4621.08 BOOL  ; Flow product number code No.8 (Lane 1)
4621.09 BOOL  ; Flow product number code No.9 (Lane 1)
4622 CHANNEL  ; Flow product number (Lane 2)
4622.01 BOOL  ; Flow product number code No.1 (Lane 2)
4622.02 BOOL  ; Flow product number code No.2 (Lane 2)
4622.03 BOOL  ; Flow product number code No.3 (Lane 2)
4622.04 BOOL  ; Flow product number code No.4 (Lane 2)
4622.05 BOOL  ; Flow product number code No.5 (Lane 2)
4622.06 BOOL  ; Flow product number code No.6 (Lane 2)
4622.07 BOOL  ; Flow product number code No.7 (Lane 2)
4622.08 BOOL  ; Flow product number code No.8 (Lane 2)
4622.09 BOOL  ; Flow product number code No.9 (Lane 2)
4623.01 BOOL  ; Code No.1 fraction workpieces having
4623.02 BOOL  ; Code No.2 fraction workpieces having
4623.03 BOOL  ; Code No.3 fraction workpieces having
4623.04 BOOL  ; Code No.4 fraction workpieces having
4623.05 BOOL  ; Code No.5 fraction workpieces having
4623.06 BOOL  ; Code No.6 fraction workpieces having
4623.07 BOOL  ; Code No.7 fraction workpieces having
4623.08 BOOL  ; Code No.8 fraction workpieces having
4623.09 BOOL  ; Code No.9 fraction workpieces having
4624 CHANNEL  ; Unloading robot workpiece code
4624.01 BOOL  ; Unloading robot workpiece code No.1
4624.02 BOOL  ; Unloading robot workpiece code No.2
4624.03 BOOL  ; Unloading robot workpiece code No.3
4624.04 BOOL  ; Unloading robot workpiece code No.4
4624.05 BOOL  ; Unloading robot workpiece code No.5
4624.06 BOOL  ; Unloading robot workpiece code No.6
4624.07 BOOL  ; Unloading robot workpiece code No.7
4624.08 BOOL  ; Unloading robot workpiece code No.8
4624.09 BOOL  ; Unloading robot workpiece code No.9
4625 CHANNEL  ; Code No. switch
4625.01 BOOL  ; Code No.1 switch
4625.02 BOOL  ; Code No.2 switch
4625.03 BOOL  ; Code No.3 switch
4625.04 BOOL  ; Code No.4 switch
4625.05 BOOL  ; Code No.5 switch
4625.06 BOOL  ; Code No.6 switch
4625.07 BOOL  ; Code No.7 switch
4625.08 BOOL  ; Code No.8 switch
4625.09 BOOL  ; Code No.9 switch
4626 CHANNEL  ; Next product number code (Lane 1)
4626.01 BOOL  ; Next product number code No.1 (Lane 1)
4626.02 BOOL  ; Next product number code No.2 (Lane 1)
4626.03 BOOL  ; Next product number code No.3 (Lane 1)
4626.04 BOOL  ; Next product number code No.4 (Lane 1)
4626.05 BOOL  ; Next product number code No.5 (Lane 1)
4626.06 BOOL  ; Next product number code No.6 (Lane 1)
4626.07 BOOL  ; Next product number code No.7 (Lane 1)
4626.08 BOOL  ; Next product number code No.8 (Lane 1)
4626.09 BOOL  ; Next product number code No.9 (Lane 1)
4627 CHANNEL  ; Next product number code (Lane 2)
4627.01 BOOL  ; Next product number code No.1 (Lane 2)
4627.02 BOOL  ; Next product number code No.2 (Lane 2)
4627.03 BOOL  ; Next product number code No.3 (Lane 2)
4627.04 BOOL  ; Next product number code No.4 (Lane 2)
4627.05 BOOL  ; Next product number code No.5 (Lane 2)
4627.06 BOOL  ; Next product number code No.6 (Lane 2)
4627.07 BOOL  ; Next product number code No.7 (Lane 2)
4627.08 BOOL  ; Next product number code No.8 (Lane 2)
4627.09 BOOL  ; Next product number code No.9 (Lane 2)
4630.00 BOOL  ; UNLOADING ROBOT CHUCK CLAMP
4630.01 BOOL  ; UNLOADING ROBOT CHUCK UNCLAMP
4631.01 BOOL  ; ROBOT START
4633.04 BOOL  ; 排出ﾛｰﾀﾞ前後_NGスタンプ位置１へ移動
4633.05 BOOL  ; 排出ﾛｰﾀﾞ前後_NGスタンプ位置2へ移動
4633.06 BOOL  ; 排出ﾛｰﾀﾞ前後_NGスタンプ位置3へ移動
4633.07 BOOL  ; 排出ﾛｰﾀﾞ前後_NGスタンプ位置4へ移動
4633.08 BOOL  ; 排出ﾛｰﾀﾞ前後_NGスタンプ位置5へ移動
4633.15 BOOL  ; 排出ﾛｰﾀﾞNGどれでもない
4634.01 BOOL  ; Fraction workpiece discharge (Lane 1)
4634.02 BOOL  ; Fraction workpiece discharge (Lane 2)
4634.03 BOOL  ; Selection of number at taking out positions of fraction workpiece
4634.04 BOOL  ; ...code No.1 fraction workpiece.. taking out
4634.05 BOOL  ; ...code No.2 fraction workpiece.. taking out
4634.06 BOOL  ; ...code No.3 fraction workpiece.. taking out
4634.07 BOOL  ; ...code No.4 fraction workpiece.. taking out
4634.08 BOOL  ; ...code No.5 fraction workpiece.. taking out
4634.09 BOOL  ; ...code No.6 fraction workpiece.. taking out
4634.10 BOOL  ; ...code No.7 fraction workpiece.. taking out
4634.11 BOOL  ; ...code No.8 fraction workpiece.. taking out
4634.12 BOOL  ; ...code No.9 fraction workpiece.. taking out
4634.13 BOOL  ; The fraction workpiece is  discharged
4634.14 BOOL  ; End of selection of number at taking out positions of fraction workpiece
4635.01 BOOL  ; The fraction workpiece is  discharged (Lane 1)
4635.02 BOOL  ; The fraction workpiece is  discharged (Lane 2)
4636.00 BOOL  ; Selection of positional number of workpiece discharge
4636.01 BOOL  ; The workpiece of the unloading robot is a good product
4636.02 BOOL  ; Workpiece discharge to lane 1
4636.03 BOOL  ; Workpiece discharge to lane 2
4636.04 BOOL  ; Workpiece discharge to lane 1 (to exchange container)
4636.05 BOOL  ; Workpiece discharge to lane 2 (to exchange container)
4636.06 BOOL  ; Workpiece discharge to lane 1 (to container befor exchange)
4636.07 BOOL  ; Workpiece discharge to lane 2 (to container befor exchange)
4636.08 BOOL  ; Fraction workpiece can be exhausted to the container
4636.09 BOOL  ; Fraction workpiece container discharge
4636.10 BOOL  ; Defective exhaust C/V discharge
4636.11 BOOL  ; End of selection of positional number of workpiece discharge
4637.01 BOOL  ; Switch of product number of lane 1
4637.02 BOOL  ; Switch of product number of lane 2
4637.03 BOOL  ; There is no switch next product number
4637.04 BOOL  ; Full workpieces of fraction workpiece container
4637.05 BOOL  ; The fraction workpiece is  discharged
4637.06 BOOL  ; Disagreement of product number (Lane 1 to exchange container)
4637.07 BOOL  ; Disagreement of product number (Lane 2 to exchange container)
4637.08 BOOL  ; Disagreement of product number (Lane 1 to  container befor exchange)
4637.09 BOOL  ; Disagreement of product number (Lane 2 to  container befor exchange)
4640.00 BOOL  ; UNLOADING ROBOT CHUCK CLAMP
4640.01 BOOL  ; UNLOADING ROBOT CHUCK UNCLAMP
4640.04 BOOL  ; Start of the fraction workpiece is discharged
4643.01 BOOL  ; ...taking out.. start acceptance of workpiece
4643.02 BOOL  ; Transfer-carrier backward signal receipt
4643.10 BOOL  ; The fraction workpiece is  discharged
4645.00 BOOL  ; 11ST_HOME POSITION
4645.01 BOOL  ; 11ST_CYCLE RUNNING
4646.01 BOOL  ; Exchange of containers (Lane 1 to exchange container)
4646.02 BOOL  ; Exchange of containers (Lane 1 to container befor exchange)
4646.03 BOOL  ; Exchange of containers (Lane 1 to exchange container)
4646.04 BOOL  ; Exchange of containers (Lane 1 to container befor exchange)
4647.01 BOOL  ; Exchange of containers (Lane 2 to exchange container)
4647.02 BOOL  ; Exchange of containers (Lane 2 to container befor exchange)
4647.03 BOOL  ; Exchange of containers (Lane 2 to exchange container)
4647.04 BOOL  ; Exchange of containers (Lane 2 to container befor exchange)
4653.00 BOOL  ; 12ST_1CY START PB on
4653.01 BOOL  ; 12ST_1CY RUN
4653.02 BOOL  ; 12ST_INDIV STEP START
4653.03 BOOL  ; 12ST_UNIT HOME POSITION PB
4653.04 BOOL  ; 12ST_UNIT HOME POSITION PB PLUSE
4654.00 BOOL  ; 12ST_CONDITION OF START(AUTO)
4654.01 BOOL  ; 12ST_CONDITION OF START(INDIV)
4654.04 BOOL  ; 12ST_CONDITION OF CYCLE START
4654.08 BOOL  ; 12ST_START RESET
4654.09 BOOL  ; 12ST_STEP UP ENABLE
4655.00 BOOL  ; 12ST_CYCLE RUNNING
4655.01 BOOL  ; 12ST_CYCLE RUNNING PLUSE
4655.02 BOOL  ; 12ST_STEP UP ENABLE
4655.03 BOOL  ; BEARING SUPPLY START
4655.04 BOOL  ; BEARING TRANSFER START
4655.15 BOOL  ; 12ST_CYCLE COMPLETE
4680.00 BOOL  ; BEARING TRANSFER CARRIER FORWARD
4680.01 BOOL  ; BEARING TRANSFER CARRIER BACKWARD
4680.02 BOOL  ; BEARING SUPPLY ROBOT TAKING OUT POSITION
4680.03 BOOL  ; BEARING SUPPLY ROBOT HOME POSITION
4680.04 BOOL  ; BEARING HANGER FORWARD
4680.05 BOOL  ; BEARING HANGER BACKWARD
4680.06 BOOL  ; BEARING HANGER DOWNWARD
4680.07 BOOL  ; BEARING HANGER UPWARD
4680.08 BOOL  ; BEARING TRANSFER UPWARD
4680.09 BOOL  ; BEARING TRANSFER DOWNWARD
4680.10 BOOL  ; BEARING PUSHER BACKWARD
4680.11 BOOL  ; BEARING PUSHER FORWARD
4680.15 BOOL  ; BEARING TRANSFER DOWNWARD
4690.00 BOOL  ; BEARING TRANSFER CARRIER FORWARD
4690.01 BOOL  ; BEARING TRANSFER CARRIER BACKWARD
4690.02 BOOL  ; BEARING SUPPLY ROBOT TAKING OUT POSITION
4690.03 BOOL  ; BEARING SUPPLY ROBOT HOME POSITION
4690.04 BOOL  ; BEARING HANGER FORWARD
4690.05 BOOL  ; BEARING HANGER BACKWARD
4690.06 BOOL  ; BEARING HANGER DOWNWARD
4690.07 BOOL  ; BEARING HANGER UPWARD
4690.08 BOOL  ; BEARING TRANSFER UPWARD
4690.09 BOOL  ; BEARING TRANSFER DOWNWARD
4690.10 BOOL  ; BEARING PUSHER BACKWARD
4690.11 BOOL  ; BEARING PUSHER FORWARD
4695.00 BOOL  ; 12ST_HOME POSITION
4695.01 BOOL  ; 12ST_CYCLE RUNNING
4702.00 BOOL  ; Exchange signal of baring tray
4702.03 BOOL  ; NO INTERFERENCE OF BEARING SUPPLY ROBOT
4703.00 BOOL  ; 13ST_1CY START PB on
4703.01 BOOL  ; 13ST_1CY RUN
4703.02 BOOL  ; 13ST_INDIV STEP START
4703.03 BOOL  ; 13ST_UNIT HOME POSITION PB
4703.04 BOOL  ; 13ST_UNIT HOME POSITION PB PLUSE
4704.00 BOOL  ; 13ST_CONDITION OF START(AUTO)
4704.01 BOOL  ; 13ST_CONDITION OF START(INDIV)
4704.04 BOOL  ; 13ST_CONDITION OF CYCLE START
4704.08 BOOL  ; 13ST_START RESET
4704.09 BOOL  ; 13ST_STEP UP ENABLE
4705.00 BOOL  ; 13ST_CYCLE RUNNING
4705.01 BOOL  ; 13ST_CYCLE RUNNING PLUSE
4705.02 BOOL  ; 13ST_STEP UP ENABLE
4705.03 BOOL  ; Unloading tray sending start
4705.04 BOOL  ; Start without tray
4705.05 BOOL  ; Tray exchange start
4705.06 BOOL  ; Loading tray sending start
4705.15 BOOL  ; 13ST_CYCLE COMPLETE
4730.00 BOOL  ; BEARING TRAY HOME POSITIONING FORWARD
4730.01 BOOL  ; BEARING TRAY HOME POSITIONING BACKWARD
4730.02 BOOL  ; BEARING TRAY EXCHANGE DOWNWARD
4730.03 BOOL  ; BEARING TRAY EXCHANGE UPWARD
4730.04 BOOL  ; BEARING TRAY STOPPER BACKWARD
4730.05 BOOL  ; BEARING TRAY STOPPER FORWARD
4730.06 BOOL  ; BEARING TRAY ESCAPE FORWARD
4730.07 BOOL  ; BEARING TRAY ESCAPE BACKWARD
4730.08 BOOL  ; EXCHANGE CONVEYOR CW ROTATE
4730.09 BOOL  ; EXCHANGE CONVEYOR CCW ROTATE
4730.12 BOOL  ; LOADING CONVEYOR ON
4730.13 BOOL  ; UNLOADING CONVEYOR ON
4731.00 BOOL  ; BEARING TRAY PASSING
4740.00 BOOL  ; BEARING TRAY HOME POSITIONING FORWARD
4740.01 BOOL  ; BEARING TRAY HOME POSITIONING BACKWARD
4740.02 BOOL  ; BEARING TRAY EXCHANGE DOWNWARD
4740.03 BOOL  ; BEARING TRAY EXCHANGE UPWARD
4740.04 BOOL  ; BEARING TRAY STOPPER BACKWARD
4740.05 BOOL  ; BEARING TRAY STOPPER FORWARD
4740.06 BOOL  ; BEARING TRAY ESCAPE FORWARD
4740.07 BOOL  ; BEARING TRAY ESCAPE BACKWARD
4740.08 BOOL  ; EXCHANGE CONVEYOR CW ROTATE
4740.09 BOOL  ; EXCHANGE CONVEYOR CCW ROTATE
4740.12 BOOL  ; LOADING CONVEYOR ON
4740.13 BOOL  ; UNLOADING CONVEYOR ON
4740.14 BOOL  ; CONVEYOR OFF
4745.00 BOOL  ; 13ST_HOME POSITION
4745.01 BOOL  ; 13ST_CYCLE RUNNING
4753.00 BOOL  ; 14ST_1CY START PB on
4753.01 BOOL  ; 14ST_1CY RUN
4753.02 BOOL  ; 14ST_INDIV STEP START
4753.03 BOOL  ; 14ST_UNIT HOME POSITION PB
4753.04 BOOL  ; 14ST_UNIT HOME POSITION PB PLUSE
4753.11 BOOL  ; FULL DEFECTS
4754.00 BOOL  ; 14ST_CONDITION OF START(AUTO)
4754.01 BOOL  ; 14ST_CONDITION OF START(INDIV)
4754.04 BOOL  ; 14ST_CONDITION OF CYCLE START
4754.08 BOOL  ; 14ST_START RESET
4754.09 BOOL  ; 14ST_STEP UP ENABLE
4755.00 BOOL  ; 14ST_CYCLE RUNNING
4755.01 BOOL  ; 14ST_CYCLE RUNNING PLUSE
4755.02 BOOL  ; 14ST_STEP UP ENABLE
4755.15 BOOL  ; 14ST_CYCLE COMPLETE
4780.00 BOOL  ; DEFECT CONVEYOR ON
4790.00 BOOL  ; DEFECT CONVEYOR ON
4790.01 BOOL  ; DEFECT CONVEYOR OFF
4795.00 BOOL  ; 14ST_HOME POSITION
4795.01 BOOL  ; 14ST_CYCLE RUNNING
4802.00 BOOL  ; PALLETIZING STOPPER DOWNWARD SIGNAL (Lane 1)
4802.05 BOOL  ; STOP SIGNAL OF CONVEYOR AFTER PALLETIZING
4803.00 BOOL  ; 15ST_1CY START PB on
4803.01 BOOL  ; 15ST_1CY RUN
4803.02 BOOL  ; 15ST_INDIV STEP START
4803.03 BOOL  ; 15ST_UNIT HOME POSITION PB
4803.04 BOOL  ; 15ST_UNIT HOME POSITION PB PLUSE
4804.00 BOOL  ; 15ST_CONDITION 1 OF START
4804.01 BOOL  ; 15ST_CONDITION 2 OF START
4804.02 BOOL  ; 15ST_CONDITION 3 OF START
4804.03 BOOL  ; 15ST_CONDITION 4 OF START
4804.04 BOOL  ; 15ST_CONDITION OF CYCLE START
4804.08 BOOL  ; 15ST_START RESET
4804.09 BOOL  ; 15ST_STEP UP ENABLE
4805.00 BOOL  ; 15ST_CYCLE RUNNING
4805.01 BOOL  ; 15ST_CYCLE RUNNING PLUSE
4805.02 BOOL  ; 15ST_STEP UP ENABLE
4805.03 BOOL  ; There is sending operation of the palletizing end container (Lane 1)
4805.04 BOOL  ; PALLETIZING START (Lane 1)
4805.05 BOOL  ; There is sending operation of the palletizing container (Lane 1)
4805.07 BOOL  ; Sending start of loading container (Lane 1)
4805.08 BOOL  ; There is no sending operation of the palletizing container (Lane 1)
4805.15 BOOL  ; 15ST_CYCLE COMPLETE
4807.00 BOOL  ; PALLETIZING HOOK BACKWARD END
4807.01 BOOL  ; PALLETIZING HOOK FORWARD END
4807.08 BOOL  ; PALLETIZING LIFTER 1 DOWNWARD END
4807.09 BOOL  ; PALLETIZING LIFTER 1 INTERMEDIATE POSITION
4807.10 BOOL  ; PALLETIZING LIFTER 1 UPWARD END
4830.00 BOOL  ; CONVEYOR AFTER PALLETIZING
4830.02 BOOL  ; STOPPER BEFOR PALLETIZING DOWNWARD
4830.03 BOOL  ; STOPPER BEFOR PALLETIZING UPWARD
4830.04 BOOL  ; PALLETIZING HOOK BACKWARD
4830.05 BOOL  ; PALLETIZING HOOK FORWARD
4830.06 BOOL  ; PALLETIZING LIFTER DOWNWARD
4830.07 BOOL  ; PALLETIZING LIFTER UPWARD
4830.08 BOOL  ; PALLETIZING CONVEYOR
4830.10 BOOL  ; STOPPER BEFOR PALLETIZING DOWNWARD
4830.11 BOOL  ; STOPPER BEFOR PALLETIZING UPWARD
4830.12 BOOL  ; LOADING CONVEYOR
4830.14 BOOL  ; ESCAPE BEFOR PALLETIZING UPWARD
4830.15 BOOL  ; ESCAPE BEFOR PALLETIZING DOWNWARD
4840.00 BOOL  ; CONVEYOR AFTER PALLETIZING
4840.01 BOOL  ; CONVEYOR STOP AFTER PALLETIZING
4840.02 BOOL  ; STOPPER BEFOR PALLETIZING DOWNWARD
4840.03 BOOL  ; STOPPER BEFOR PALLETIZING UPWARD
4840.04 BOOL  ; PALLETIZING HOOK BACKWARD
4840.05 BOOL  ; PALLETIZING HOOK FORWARD
4840.06 BOOL  ; PALLETIZING LIFTER DOWNWARD
4840.07 BOOL  ; PALLETIZING LIFTER UPWARD
4840.08 BOOL  ; PALLETIZING CONVEYOR
4840.10 BOOL  ; STOPPER BEFOR PALLETIZING DOWNWARD
4840.11 BOOL  ; STOPPER BEFOR PALLETIZING UPWARD
4840.12 BOOL  ; LOADING CONVEYOR
4840.14 BOOL  ; ESCAPE BEFOR PALLETIZING UPWARD
4840.15 BOOL  ; ESCAPE BEFOR PALLETIZING DOWNWARD
4843.01 BOOL  ; START SIGNAL OF CONVEYOR AFTER PALLETIZING
4843.05 BOOL  ; STOP SIGNAL OF CONVEYOR AFTER PALLETIZING
4845.00 BOOL  ; 15ST_HOME POSITION
4845.01 BOOL  ; 15ST_CYCLE RUNNING
4852.00 BOOL  ; Container exchange signal (container befor exchange)
4852.01 BOOL  ; CONVEYOR ROTATE AFTER PALLETIZING
4852.05 BOOL  ; CONVEYOR STOP AFTER PALLETIZING
4852.06 BOOL  ; PALLETIZING CONVEYOR STOP
4852.07 BOOL  ; Container exchange signal (exchange container)
4852.09 BOOL  ; The container exchange can operate when the product number is switched
4853.00 BOOL  ; 16ST_1CY START PB on
4853.01 BOOL  ; 16ST_1CY RUN
4853.02 BOOL  ; 16ST_INDIV STEP START
4853.03 BOOL  ; 16ST_UNIT HOME POSITION PB
4853.04 BOOL  ; 16ST_UNIT HOME POSITION PB PLUSE
4854.00 BOOL  ; 16ST_CONDITION OF START(AUTO)
4854.01 BOOL  ; 16ST_CONDITION OF START(INDIV)
4854.04 BOOL  ; 16ST_CONDITION OF CYCLE START
4854.08 BOOL  ; 16ST_START RESET
4854.09 BOOL  ; 16ST_STEP UP ENABLE
4855.00 BOOL  ; 16ST_CYCLE RUNNING
4855.01 BOOL  ; 16ST_CYCLE RUNNING PLUSE
4855.02 BOOL  ; 16ST_STEP UP ENABLE
4855.03 BOOL  ; Start without container (exchange container)
4855.04 BOOL  ; Start without container (container befor exchange )
4855.05 BOOL  ; Container exchange start
4855.12 BOOL  ; Condition waiting
4855.13 BOOL  ; Container arrival memory to palletizing unit
4855.15 BOOL  ; 16ST_CYCLE COMPLETE
4880.00 BOOL  ; POSITIONING 1 BACKWARD
4880.01 BOOL  ; POSITIONING 1 FORWARD
4880.02 BOOL  ; LIFTER DOWNWARD
4880.03 BOOL  ; LIFTER UPWARD
4880.04 BOOL  ; POSITIONING 2 BACKWARD
4880.05 BOOL  ; POSITIONING 2 FORWARD
4880.06 BOOL  ; DROP GUARD BACKWARD
4880.07 BOOL  ; DROP GUARD FORWARD
4880.08 BOOL  ; EXCHANGE CONVEYOR CW
4880.09 BOOL  ; EXCHANGE CONVEYOR CCW
4880.12 BOOL  ; PALLETIZING CONVEYOR
4880.13 BOOL  ; STACKING CONVEYOR
4890.00 BOOL  ; POSITIONING 1 BACKWARD
4890.01 BOOL  ; POSITIONING 1 FORWARD
4890.02 BOOL  ; LIFTER DOWNWARD
4890.03 BOOL  ; LIFTER UPWARD
4890.04 BOOL  ; POSITIONING 2 BACKWARD
4890.05 BOOL  ; POSITIONING 2 FORWARD
4890.06 BOOL  ; DROP GUARD BACKWARD
4890.07 BOOL  ; DROP GUARD FORWARD
4890.08 BOOL  ; EXCHANGE CONVEYOR CW
4890.09 BOOL  ; EXCHANGE CONVEYOR CCW
4890.10 BOOL  ; Writing of ID1
4890.11 BOOL  ; Writing of ID2
4890.12 BOOL  ; PALLETIZING CONVEYOR
4890.13 BOOL  ; STACKING CONVEYOR
4890.14 BOOL  ; CONVEYOR STOP
4893.00 BOOL  ; STOPPER DOWNWARD SIGNAL
4893.01 BOOL  ; Writing signal of ID1
4893.02 BOOL  ; Writing signal of ID2
4893.03 BOOL  ; STACKING CONVEYOR START SIGNAL
4893.05 BOOL  ; PALLETIZING CONVEYOR STOP SIGNAL
4893.06 BOOL  ; ﾚｰﾝ1段積み部ｺﾝﾍﾞｱ停止信号
4895.00 BOOL  ; 16ST_HOME POSITION
4895.01 BOOL  ; 16ST_CYCLE RUNNING
4902.03 BOOL  ; STACKING CONVEYOR START SIGNAL
4902.06 BOOL  ; STACKING CONVEYOR STOP SIGNAL
4902.07 BOOL  ; STACKING IMPROPRIETY
4902.08 BOOL  ; Downward confirmation when product number is switched
4902.10 BOOL  ; Disbursement completion of fraction workpiece
4903.00 BOOL  ; 17ST_1CY START PB on
4903.01 BOOL  ; 17ST_1CY RUN
4903.02 BOOL  ; 17ST_INDIV STEP START
4903.03 BOOL  ; 17ST_UNIT HOME POSITION PB
4903.04 BOOL  ; 17ST_UNIT HOME POSITION PB PLUSE
4904.00 BOOL  ; 17ST_CONDITION OF START(AUTO)
4904.01 BOOL  ; 17ST_CONDITION OF START(INDIV)
4904.04 BOOL  ; 17ST_CONDITION OF CYCLE START
4904.08 BOOL  ; 17ST_START RESET
4904.09 BOOL  ; 17ST_STEP UP ENABLE
4905.00 BOOL  ; 17ST_CYCLE RUNNING
4905.01 BOOL  ; 17ST_CYCLE RUNNING PLUSE
4905.02 BOOL  ; 17ST_STEP UP ENABLE
4905.03 BOOL  ; UNLOADING UNIT START
4905.04 BOOL  ; STACKING START
4905.05 BOOL  ; UNLOADING  START OF STACKING CONTAINER
4905.06 BOOL  ; UNLOADING PALLET CONVEYOR
4905.15 BOOL  ; 17ST_CYCLE COMPLETE
4906.08 BOOL  ; UNLOADING CONVEYOR 1
4906.12 BOOL  ; UNLOADING CONVEYOR 2
4906.13 BOOL  ; UNLOADING UNIT STOP
4907.00 BOOL  ; STACKING HOOK BACKWARD END
4907.01 BOOL  ; STACKING HOOK FORWARD END
4907.08 BOOL  ; STACKING LIFTER DOWNWARD END
4907.09 BOOL  ; STACKING LIFTER UPWARD END
4907.10 BOOL  ; STACKING LIFTER INTERMEDIATE POSITION
4930.00 BOOL  ; STACKING HOOK BACKWARD
4930.01 BOOL  ; STACKING HOOK FORWARD
4930.02 BOOL  ; STACKING LIFTER DOWNWARD
4930.03 BOOL  ; STACKING LIFTER UPWARD
4930.04 BOOL  ; STACKING CONVEYOR
4930.06 BOOL  ; STACKING STOPPER DOWNWARD
4930.07 BOOL  ; STACKING STOPPER UPWARD
4930.08 BOOL  ; UNLOADING CONVEYOR 1
4930.10 BOOL  ; UNLOADING ESCAPE UPWARD
4930.11 BOOL  ; UNLOADING ESCAPE DOWNWARD
4930.12 BOOL  ; UNLOADING CONVEYOR 2
4930.14 BOOL  ; UNLOADING STOPPER DOWNWARD
4930.15 BOOL  ; UNLOADING STOPPER UPWARD
4940.00 BOOL  ; STACKING HOOK BACKWARD
4940.01 BOOL  ; STACKING HOOK FORWARD
4940.02 BOOL  ; STACKING LIFTER DOWNWARD
4940.03 BOOL  ; STACKING LIFTER UPWARD
4940.04 BOOL  ; STACKING CONVEYOR
4940.05 BOOL  ; CONVEYOR STOP
4940.06 BOOL  ; STACKING STOPPER DOWNWARD
4940.07 BOOL  ; STACKING STOPPER UPWARD
4940.08 BOOL  ; UNLOADING CONVEYOR 1
4940.10 BOOL  ; UNLOADING ESCAPE UPWARD
4940.11 BOOL  ; UNLOADING ESCAPE DOWNWARD
4940.12 BOOL  ; UNLOADING CONVEYOR 2
4940.14 BOOL  ; UNLOADING STOPPER DOWNWARD
4940.15 BOOL  ; UNLOADING STOPPER UPWARD
4943.06 BOOL  ; STACKING CONVEYOR STOP SIGNAL
4943.07 BOOL  ; Container discharge completion
4943.08 BOOL  ; Stacking containers cannot be exchanged
4945.00 BOOL  ; 17ST_HOME POSITION
4945.01 BOOL  ; 17ST_CYCLE RUNNING
4952.00 BOOL  ; PALLETIZING STOPPER DOWNWARD SIGNAL (Lane 2)
4952.05 BOOL  ; STOP SIGNAL OF CONVEYOR AFTER PALLETIZING
4953.00 BOOL  ; 18ST_1CY START PB on
4953.01 BOOL  ; 18ST_1CY RUN
4953.02 BOOL  ; 18ST_INDIV STEP START
4953.03 BOOL  ; 18ST_UNIT HOME POSITION PB
4953.04 BOOL  ; 18ST_UNIT HOME POSITION PB PLUSE
4954.00 BOOL  ; 18ST_CONDITION 1 OF START
4954.01 BOOL  ; 18ST_CONDITION 2 OF START
4954.02 BOOL  ; 18ST_CONDITION 3 OF START
4954.03 BOOL  ; 18ST_CONDITION 4 OF START
4954.04 BOOL  ; 18ST_CONDITION OF CYCLE START
4954.08 BOOL  ; 18ST_START RESET
4954.09 BOOL  ; 18ST_STEP UP ENABLE
4955.00 BOOL  ; 18ST_CYCLE RUNNING
4955.01 BOOL  ; 18ST_CYCLE RUNNING PLUSE
4955.02 BOOL  ; 18ST_STEP UP ENABLE
4955.03 BOOL  ; There is sending operation of the palletizing end container (Lane 2)
4955.04 BOOL  ; PALLETIZING START (Lane 2)
4955.05 BOOL  ; There is sending operation of the palletizing container (Lane 2)
4955.07 BOOL  ; Sending start of loading container (Lane 2)
4955.08 BOOL  ; There is no sending operation of the palletizing container (Lane 2)
4955.15 BOOL  ; 18ST_CYCLE COMPLETE
4957.00 BOOL  ; PALLETIZING HOOK BACKWARD END
4957.01 BOOL  ; PALLETIZING HOOK FORWARD END
4957.08 BOOL  ; PALLETIZING LIFTER 2 DOWNWARD END
4957.09 BOOL  ; PALLETIZING LIFTER 2 INTERMEDIATE POSITION
4957.10 BOOL  ; PALLETIZING LIFTER 2 UPWARD END
4980.00 BOOL  ; CONVEYOR AFTER PALLETIZING
4980.02 BOOL  ; STOPPER BEFOR PALLETIZING DOWNWARD
4980.03 BOOL  ; STOPPER BEFOR PALLETIZING UPWARD
4980.04 BOOL  ; PALLETIZING HOOK BACKWARD
4980.05 BOOL  ; PALLETIZING HOOK FORWARD
4980.06 BOOL  ; PALLETIZING LIFTER DOWNWARD
4980.07 BOOL  ; PALLETIZING LIFTER UPWARD
4980.08 BOOL  ; PALLETIZING CONVEYOR
4980.10 BOOL  ; STOPPER BEFOR PALLETIZING DOWNWARD
4980.11 BOOL  ; STOPPER BEFOR PALLETIZING UPWARD
4980.12 BOOL  ; LOADING CONVEYOR
4980.14 BOOL  ; ESCAPE BEFOR PALLETIZING UPWARD
4980.15 BOOL  ; ESCAPE BEFOR PALLETIZING DOWNWARD
4990.00 BOOL  ; CONVEYOR AFTER PALLETIZING
4990.01 BOOL  ; CONVEYOR STOP AFTER PALLETIZING
4990.02 BOOL  ; STOPPER BEFOR PALLETIZING DOWNWARD
4990.03 BOOL  ; STOPPER BEFOR PALLETIZING UPWARD
4990.04 BOOL  ; PALLETIZING HOOK BACKWARD
4990.05 BOOL  ; PALLETIZING HOOK FORWARD
4990.06 BOOL  ; PALLETIZING LIFTER DOWNWARD
4990.07 BOOL  ; PALLETIZING LIFTER UPWARD
4990.08 BOOL  ; PALLETIZING CONVEYOR
4990.10 BOOL  ; STOPPER BEFOR PALLETIZING DOWNWARD
4990.11 BOOL  ; STOPPER BEFOR PALLETIZING UPWARD
4990.12 BOOL  ; LOADING CONVEYOR
4990.14 BOOL  ; ESCAPE BEFOR PALLETIZING UPWARD
4990.15 BOOL  ; ESCAPE BEFOR PALLETIZING DOWNWARD
4993.01 BOOL  ; START SIGNAL OF CONVEYOR AFTER PALLETIZING
4993.05 BOOL  ; STOP SIGNAL OF CONVEYOR AFTER PALLETIZING
4995.00 BOOL  ; 18ST_HOME POSITION
4995.01 BOOL  ; 18ST_CYCLE RUNNING
5 CHANNEL  ; RESISTANCE MEASURED VALUE
5002.00 BOOL  ; Container exchange signal (container befor exchange)
5002.01 BOOL  ; CONVEYOR ROTATE AFTER PALLETIZING
5002.05 BOOL  ; CONVEYOR STOP AFTER PALLETIZING
5002.06 BOOL  ; PALLETIZING CONVEYOR STOP
5002.07 BOOL  ; Container exchange signal (exchange container)
5002.09 BOOL  ; The container exchange can operate when the product number is switched
5003.00 BOOL  ; 19ST_1CY START PB on
5003.01 BOOL  ; 19ST_1CY RUN
5003.02 BOOL  ; 19ST_INDIV STEP START
5003.03 BOOL  ; 19ST_UNIT HOME POSITION PB
5003.04 BOOL  ; 19ST_UNIT HOME POSITION PB PLUSE
5004.00 BOOL  ; 19ST_CONDITION OF START(AUTO)
5004.01 BOOL  ; 19ST_CONDITION OF START(INDIV)
5004.04 BOOL  ; 19ST_CONDITION OF CYCLE START
5004.08 BOOL  ; 19ST_START RESET
5004.09 BOOL  ; 19ST_STEP UP ENABLE
5005.00 BOOL  ; 19ST_CYCLE RUNNING
5005.01 BOOL  ; 19ST_CYCLE RUNNING PLUSE
5005.02 BOOL  ; 19ST_STEP UP ENABLE
5005.03 BOOL  ; Start without container (exchange container)
5005.04 BOOL  ; Start without container (container befor exchange )
5005.05 BOOL  ; Container exchange start
5005.12 BOOL  ; Condition waiting
5005.13 BOOL  ; Container arrival memory to palletizing unit
5005.15 BOOL  ; 19ST_CYCLE COMPLETE
5030.00 BOOL  ; POSITIONING 1 BACKWARD
5030.01 BOOL  ; POSITIONING 1 FORWARD
5030.02 BOOL  ; LIFTER DOWNWARD
5030.03 BOOL  ; LIFTER UPWARD
5030.04 BOOL  ; POSITIONING 2 BACKWARD
5030.05 BOOL  ; POSITIONING 2 FORWARD
5030.06 BOOL  ; DROP GUARD BACKWARD
